LIN {X 0,Y 317.78,Z 749.574,A -85,B 0,C 180,E1 -15963.012,E2 -15963.012} C_VEL
LIN {X 0,Y 315.346,Z 742.44,A -85,B 0,C 180,E1 -15964.324,E2 -15964.324} C_VEL
LIN {X 0,Y 313.028,Z 732.738,A -85,B 0,C 180,E1 -15966.631,E2 -15966.631} C_VEL
LIN {X 0,Y 311.777,Z 725.359,A -85,B 0,C 180,E1 -15968.715,E2 -15968.715} C_VEL
LIN {X 0,Y 311.359,Z 724.12,A -85,B 0,C 180,E1 -15969.207,E2 -15969.207} C_VEL
LIN {X 0,Y 309.328,Z 721.332,A -85,B 0,C 180,E1 -15971.223,E2 -15971.223} C_VEL
LIN {X 0,Y 308.008,Z 719.093,A -85,B 0,C 180,E1 -15973.207,E2 -15973.207} C_VEL
LIN {X 0,Y 306.578,Z 717.561,A -85,B 0,C 180,E1 -15976.55,E2 -15976.55} C_VEL
LIN {X 0,Y 306.472,Z 717.374,A -85,B 0,C 180,E1 -15979.188,E2 -15979.188} C_VEL
LIN {X 0,Y 307.274,Z 718.36,A -85,B 0,C 180,E1 -15982.108,E2 -15982.108} C_VEL
LIN {X 0,Y 310.182,Z 720.574,A -85,B 0,C 180,E1 -15984.209,E2 -15984.209} C_VEL
LIN {X 0,Y 311.655,Z 723.597,A -85,B 0,C 180,E1 -15985.294,E2 -15985.294} C_VEL
LIN {X 0,Y 314.049,Z 725.859,A -85,B 0,C 180,E1 -15986.519,E2 -15986.519} C_VEL
LIN {X 0,Y 315.86,Z 729.038,A -85,B 0,C 180,E1 -15987.472,E2 -15987.472} C_VEL
LIN {X 0,Y 317.513,Z 730.978,A -85,B 0,C 180,E1 -15988.203,E2 -15988.203} C_VEL
LIN {X 0,Y 320.745,Z 736.046,A -85,B 0,C 180,E1 -15989.561,E2 -15989.561} C_VEL
LIN {X 0,Y 323.632,Z 740.623,A -85,B 0,C 180,E1 -15990.632,E2 -15990.632} C_VEL
LIN {X 0,Y 328.07,Z 748.441,A -85,B 0,C 180,E1 -15992.144,E2 -15992.144} C_VEL
LIN {X 0,Y 330.075,Z 752.544,A -85,B 0,C 180,E1 -15992.8,E2 -15992.8} C_VEL
LIN {X 0,Y 326.244,Z 796.508,A -85,B 0,C 180,E1 -15994.522,E2 -15994.522} C_VEL
LIN {X 0,Y 325.441,Z 812.458,A -85,B 0,C 180,E1 -15995.266,E2 -15995.266} C_VEL
LIN {X 0,Y 324.627,Z 823.18,A -85,B 0,C 180,E1 -15995.929,E2 -15995.929} C_VEL
LIN {X 0,Y 323.492,Z 834.349,A -85,B 0,C 180,E1 -15996.818,E2 -15996.818} C_VEL
LIN {X 0,Y 321.89,Z 846.494,A -85,B 0,C 180,E1 -15998.044,E2 -15998.044} C_VEL
LIN {X 0,Y 320.226,Z 856.26,A -85,B 0,C 180,E1 -15999.274,E2 -15999.274} C_VEL
LIN {X 0,Y 318.57,Z 865.22,A -85,B 0,C 180,E1 -16000.676,E2 -16000.676} C_VEL
LIN {X 0,Y 317.098,Z 871.96,A -85,B 0,C 180,E1 -16001.923,E2 -16001.923} C_VEL
LIN {X 0,Y 315.396,Z 879.003,A -85,B 0,C 180,E1 -16003.477,E2 -16003.477} C_VEL
LIN {X 0,Y 313.824,Z 884.946,A -85,B 0,C 180,E1 -16005.076,E2 -16005.076} C_VEL
LIN {X 0,Y 312.104,Z 890.624,A -85,B 0,C 180,E1 -16006.986,E2 -16006.986} C_VEL
LIN {X 0,Y 311.032,Z 893.718,A -85,B 0,C 180,E1 -16008.266,E2 -16008.266} C_VEL
LIN {X 0,Y 310.152,Z 896.329,A -85,B 0,C 180,E1 -16009.556,E2 -16009.556} C_VEL
LIN {X 0,Y 308.48,Z 899.873,A -85,B 0,C 180,E1 -16012.143,E2 -16012.143} C_VEL
LIN {X 0,Y 307.923,Z 901.043,A -85,B 0,C 180,E1 -16013.447,E2 -16013.447} C_VEL
LIN {X 0,Y 307.007,Z 901.892,A -85,B 0,C 180,E1 -16016.062,E2 -16016.062} C_VEL
LIN {X 0,Y 306.544,Z 901.716,A -85,B 0,C 180,E1 -16017.372,E2 -16017.372} C_VEL
LIN {X 0,Y 306.293,Z 901.04,A -85,B 0,C 180,E1 -16018.685,E2 -16018.685} C_VEL
LIN {X 0,Y 305.877,Z 899.917,A -85,B 0,C 180,E1 -16020,E2 -16020} C_VEL
LIN {X 0,Y 305.848,Z 898.443,A -85,B 0,C 180,E1 -16021.317,E2 -16021.317} C_VEL
LIN {X 0,Y 305.552,Z 895.298,A -85,B 0,C 180,E1 -16023.297,E2 -16023.297} C_VEL
LIN {X 0,Y 305.718,Z 891.017,A -85,B 0,C 180,E1 -16025.276,E2 -16025.276} C_VEL
LIN {X 0,Y 306.118,Z 885.522,A -85,B 0,C 180,E1 -16027.254,E2 -16027.254} C_VEL
LIN {X 0,Y 306.415,Z 879.941,A -85,B 0,C 180,E1 -16028.906,E2 -16028.906} C_VEL
LIN {X 0,Y 306.759,Z 873.225,A -85,B 0,C 180,E1 -16030.561,E2 -16030.561} C_VEL
LIN {X 0,Y 307.31,Z 865.158,A -85,B 0,C 180,E1 -16032.213,E2 -16032.213} C_VEL
LIN {X 0,Y 307.837,Z 856.481,A -85,B 0,C 180,E1 -16033.702,E2 -16033.702} C_VEL
LIN {X 0,Y 308.322,Z 848.553,A -85,B 0,C 180,E1 -16034.859,E2 -16034.859} C_VEL
LIN {X 0,Y 308.959,Z 839.214,A -85,B 0,C 180,E1 -16036.011,E2 -16036.011} C_VEL
LIN {X 0,Y 309.468,Z 829.618,A -85,B 0,C 180,E1 -16037.001,E2 -16037.001} C_VEL
LIN {X 0,Y 309.947,Z 818.852,A -85,B 0,C 180,E1 -16037.909,E2 -16037.909} C_VEL
LIN {X 0,Y 310.257,Z 809.036,A -85,B 0,C 180,E1 -16038.575,E2 -16038.575} C_VEL
LIN {X 0,Y 310.505,Z 798.799,A -85,B 0,C 180,E1 -16039.117,E2 -16039.117} C_VEL
LIN {X 0,Y 310.764,Z 784.432,A -85,B 0,C 180,E1 -16039.658,E2 -16039.658} C_VEL
LIN {X 0,Y 311.932,Z 734.903,A -85,B 0,C 180,E1 -16041.245,E2 -16041.245} C_VEL
LIN {X 0,Y 305.553,Z 714.421,A -85,B 0,C 180,E1 -16042.227,E2 -16042.227} C_VEL
LIN {X 0,Y 305.492,Z 714.43,A -85,B 0,C 180,E1 -16046.194,E2 -16046.194} C_VEL
LIN {X 0,Y 305.459,Z 714.438,A -85,B 0,C 180,E1 -16049.026,E2 -16049.026} C_VEL
LIN {X 0,Y 305.459,Z 714.434,A -85,B 0,C 180,E1 -16051.951,E2 -16051.951} C_VEL
LIN {X 0,Y 305.483,Z 714.432,A -85,B 0,C 180,E1 -16055.111,E2 -16055.111} C_VEL
LIN {X 0,Y 305.457,Z 714.434,A -85,B 0,C 180,E1 -16058.521,E2 -16058.521} C_VEL
LIN {X 0,Y 305.455,Z 714.432,A -85,B 0,C 180,E1 -16062.577,E2 -16062.577} C_VEL
LIN {X 0,Y 305.441,Z 714.431,A -85,B 0,C 180,E1 -16066.339,E2 -16066.339} C_VEL
LIN {X 0,Y 305.431,Z 714.433,A -85,B 0,C 180,E1 -16069.88,E2 -16069.88} C_VEL
LIN {X 0,Y 305.481,Z 714.427,A -85,B 0,C 180,E1 -16073.632,E2 -16073.632} C_VEL
LIN {X 0,Y 305.483,Z 714.427,A -85,B 0,C 180,E1 -16076.478,E2 -16076.478} C_VEL
LIN {X 0,Y 305.431,Z 714.436,A -85,B 0,C 180,E1 -16079.58,E2 -16079.58} C_VEL
LIN {X 0,Y 305.457,Z 714.431,A -85,B 0,C 180,E1 -16082.595,E2 -16082.595} C_VEL
LIN {X 0,Y 305.493,Z 714.428,A -85,B 0,C 180,E1 -16083.931,E2 -16083.931} C_VEL
LIN {X 0,Y 306.567,Z 717.417,A -85,B 0,C 180,E1 -16084.128,E2 -16084.128} C_VEL
LIN {X 0,Y 314.491,Z 733.858,A -85,B 0,C 180,E1 -16085.267,E2 -16085.267} C_VEL
LIN {X 0,Y 318.357,Z 742.756,A -85,B 0,C 180,E1 -16085.82,E2 -16085.82} C_VEL
LIN {X 0,Y 317.568,Z 789.63,A -85,B 0,C 180,E1 -16086.896,E2 -16086.896} C_VEL
LIN {X 0,Y 317.483,Z 803.278,A -85,B 0,C 180,E1 -16087.318,E2 -16087.318} C_VEL
LIN {X 0,Y 317.084,Z 815.616,A -85,B 0,C 180,E1 -16087.943,E2 -16087.943} C_VEL
LIN {X 0,Y 316.257,Z 828.425,A -85,B 0,C 180,E1 -16088.858,E2 -16088.858} C_VEL
LIN {X 0,Y 315.223,Z 840.006,A -85,B 0,C 180,E1 -16089.957,E2 -16089.957} C_VEL
LIN {X 0,Y 313.996,Z 850.475,A -85,B 0,C 180,E1 -16091.224,E2 -16091.224} C_VEL
LIN {X 0,Y 312.703,Z 860.073,A -85,B 0,C 180,E1 -16092.667,E2 -16092.667} C_VEL
LIN {X 0,Y 311.526,Z 868.767,A -85,B 0,C 180,E1 -16094.285,E2 -16094.285} C_VEL
LIN {X 0,Y 310.053,Z 877.271,A -85,B 0,C 180,E1 -16096.223,E2 -16096.223} C_VEL
LIN {X 0,Y 308.81,Z 884.034,A -85,B 0,C 180,E1 -16098.173,E2 -16098.173} C_VEL
LIN {X 0,Y 308.073,Z 889.399,A -85,B 0,C 180,E1 -16100.14,E2 -16100.14} C_VEL
LIN {X 0,Y 307.587,Z 892.335,A -85,B 0,C 180,E1 -16101.451,E2 -16101.451} C_VEL
LIN {X 0,Y 306.655,Z 895.896,A -85,B 0,C 180,E1 -16103.412,E2 -16103.412} C_VEL
LIN {X 0,Y 306.29,Z 897.719,A -85,B 0,C 180,E1 -16104.725,E2 -16104.725} C_VEL
LIN {X 0,Y 306.079,Z 900.031,A -85,B 0,C 180,E1 -16107.359,E2 -16107.359} C_VEL
LIN {X 0,Y 305.857,Z 900.872,A -85,B 0,C 180,E1 -16109.991,E2 -16109.991} C_VEL
LIN {X 0,Y 306.079,Z 900.108,A -85,B 0,C 180,E1 -16112.623,E2 -16112.623} C_VEL
LIN {X 0,Y 306.272,Z 897.878,A -85,B 0,C 180,E1 -16115.257,E2 -16115.257} C_VEL
LIN {X 0,Y 306.892,Z 895.061,A -85,B 0,C 180,E1 -16117.227,E2 -16117.227} C_VEL
LIN {X 0,Y 307.753,Z 891.234,A -85,B 0,C 180,E1 -16119.189,E2 -16119.189} C_VEL
LIN {X 0,Y 308.611,Z 885.762,A -85,B 0,C 180,E1 -16121.358,E2 -16121.358} C_VEL
LIN {X 0,Y 309.801,Z 878.949,A -85,B 0,C 180,E1 -16123.436,E2 -16123.436} C_VEL
LIN {X 0,Y 311.214,Z 870.92,A -85,B 0,C 180,E1 -16125.377,E2 -16125.377} C_VEL
LIN {X 0,Y 312.441,Z 862.701,A -85,B 0,C 180,E1 -16126.993,E2 -16126.993} C_VEL
LIN {X 0,Y 313.765,Z 852.531,A -85,B 0,C 180,E1 -16128.603,E2 -16128.603} C_VEL
LIN {X 0,Y 315.084,Z 842.061,A -85,B 0,C 180,E1 -16129.92,E2 -16129.92} C_VEL
LIN {X 0,Y 316.183,Z 830.793,A -85,B 0,C 180,E1 -16131.048,E2 -16131.048} C_VEL
LIN {X 0,Y 317.074,Z 818.868,A -85,B 0,C 180,E1 -16131.954,E2 -16131.954} C_VEL
LIN {X 0,Y 317.491,Z 806.497,A -85,B 0,C 180,E1 -16132.646,E2 -16132.646} C_VEL
LIN {X 0,Y 317.657,Z 795.086,A -85,B 0,C 180,E1 -16133.069,E2 -16133.069} C_VEL
LIN {X 0,Y 318.132,Z 758.842,A -85,B 0,C 180,E1 -16133.922,E2 -16133.922} C_VEL
LIN {X 0,Y 318.417,Z 742.883,A -85,B 0,C 180,E1 -16134.287,E2 -16134.287} C_VEL
LIN {X 0,Y 310.461,Z 725.118,A -85,B 0,C 180,E1 -16135.431,E2 -16135.431} C_VEL
LIN {X 0,Y 305.739,Z 715.497,A -85,B 0,C 180,E1 -16136.119,E2 -16136.119} C_VEL
LIN {X 0,Y 305.504,Z 714.422,A -85,B 0,C 180,E1 -16136.21,E2 -16136.21} C_VEL
LIN {X 0,Y 305.424,Z 714.435,A -85,B 0,C 180,E1 -16140.188,E2 -16140.188} C_VEL
LIN {X 0,Y 305.433,Z 714.435,A -85,B 0,C 180,E1 -16144.069,E2 -16144.069} C_VEL
LIN {X 0,Y 305.435,Z 714.436,A -85,B 0,C 180,E1 -16145.905,E2 -16145.905} C_VEL
LIN {X 0,Y 304.811,Z 714.517,A -85,B 0,C 180,E1 -16147.006,E2 -16147.006} C_VEL
LIN {X 0,Y 301.976,Z 714.877,A -85,B 0,C 180,E1 -16148.797,E2 -16148.797} C_VEL
LIN {X 0,Y 299.539,Z 715.18,A -85,B 0,C 180,E1 -16150.251,E2 -16150.251} C_VEL
LIN {X 0,Y 298.48,Z 715.31,A -85,B 0,C 180,E1 -16151.377,E2 -16151.377} C_VEL
LIN {X 0,Y 298.389,Z 715.314,A -85,B 0,C 180,E1 -16151.758,E2 -16151.758} C_VEL
LIN {X 0,Y 298.446,Z 715.285,A -85,B 0,C 180,E1 -16155.052,E2 -16155.052} C_VEL
LIN {X 0,Y 298.407,Z 715.316,A -85,B 0,C 180,E1 -16158.89,E2 -16158.89} C_VEL
LIN {X 0,Y 298.415,Z 715.312,A -85,B 0,C 180,E1 -16163.18,E2 -16163.18} C_VEL
LIN {X 0,Y 298.343,Z 715.317,A -85,B 0,C 180,E1 -16167.193,E2 -16167.193} C_VEL
LIN {X 0,Y 298.376,Z 715.306,A -85,B 0,C 180,E1 -16170.609,E2 -16170.609} C_VEL
LIN {X 0,Y 298.421,Z 715.31,A -85,B 0,C 180,E1 -16173.471,E2 -16173.471} C_VEL
LIN {X 0,Y 298.373,Z 715.308,A -85,B 0,C 180,E1 -16176.694,E2 -16176.694} C_VEL
LIN {X 0,Y 298.476,Z 715.3,A -85,B 0,C 180,E1 -16180.752,E2 -16180.752} C_VEL
LIN {X 0,Y 298.528,Z 715.3,A -85,B 0,C 180,E1 -16184.991,E2 -16184.991} C_VEL
LIN {X 0,Y 298.527,Z 715.286,A -85,B 0,C 180,E1 -16189.144,E2 -16189.144} C_VEL
LIN {X 0,Y 298.683,Z 715.28,A -85,B 0,C 180,E1 -16191.884,E2 -16191.884} C_VEL
LIN {X 0,Y 298.595,Z 715.288,A -85,B 0,C 180,E1 -16194.598,E2 -16194.598} C_VEL
LIN {X 0,Y 298.861,Z 715.26,A -85,B 0,C 180,E1 -16198.652,E2 -16198.652} C_VEL
LIN {X 0,Y 298.861,Z 715.253,A -85,B 0,C 180,E1 -16201.347,E2 -16201.347} C_VEL
LIN {X 0,Y 298.596,Z 715.296,A -85,B 0,C 180,E1 -16205.402,E2 -16205.402} C_VEL
LIN {X 0,Y 298.683,Z 715.274,A -85,B 0,C 180,E1 -16208.116,E2 -16208.116} C_VEL
LIN {X 0,Y 298.488,Z 715.304,A -85,B 0,C 180,E1 -16212.234,E2 -16212.234} C_VEL
LIN {X 0,Y 298.521,Z 715.301,A -85,B 0,C 180,E1 -16215.198,E2 -16215.198} C_VEL
LIN {X 0,Y 298.462,Z 715.305,A -85,B 0,C 180,E1 -16219.248,E2 -16219.248} C_VEL
LIN {X 0,Y 298.395,Z 715.317,A -85,B 0,C 180,E1 -16223.603,E2 -16223.603} C_VEL
LIN {X 0,Y 298.427,Z 715.303,A -85,B 0,C 180,E1 -16226.58,E2 -16226.58} C_VEL
LIN {X 0,Y 298.365,Z 715.313,A -85,B 0,C 180,E1 -16229.647,E2 -16229.647} C_VEL
LIN {X 0,Y 298.343,Z 715.32,A -85,B 0,C 180,E1 -16232.807,E2 -16232.807} C_VEL
LIN {X 0,Y 298.415,Z 715.309,A -85,B 0,C 180,E1 -16236.82,E2 -16236.82} C_VEL
LIN {X 0,Y 298.407,Z 715.314,A -85,B 0,C 180,E1 -16241.258,E2 -16241.258} C_VEL
LIN {X 0,Y 298.446,Z 715.308,A -85,B 0,C 180,E1 -16245.069,E2 -16245.069} C_VEL
LIN {X 0,Y 298.414,Z 715.312,A -85,B 0,C 180,E1 -16248.907,E2 -16248.907} C_VEL
LIN {X 0,Y 298.416,Z 715.345,A -85,B 0,C 180,E1 -16249.765,E2 -16249.765} C_VEL
LIN {X 0,Y 301.883,Z 728.539,A -85,B 0,C 180,E1 -16253.434,E2 -16253.434} C_VEL
LIN {X 0,Y 304.482,Z 739.897,A -85,B 0,C 180,E1 -16256.374,E2 -16256.374} C_VEL
LIN {X 0,Y 306.355,Z 749.348,A -85,B 0,C 180,E1 -16258.703,E2 -16258.703} C_VEL
LIN {X 0,Y 303.364,Z 769.628,A -85,B 0,C 180,E1 -16263.081,E2 -16263.081} C_VEL
LIN {X 0,Y 307.305,Z 801.463,A -85,B 0,C 180,E1 -16264.256,E2 -16264.256} C_VEL
LIN {X 0,Y 310.222,Z 833.466,A -85,B 0,C 180,E1 -16265.3,E2 -16265.3} C_VEL
LIN {X 0,Y 308.939,Z 881.214,A -85,B 0,C 180,E1 -16266.418,E2 -16266.418} C_VEL
LIN {X 0,Y 308.109,Z 894.367,A -85,B 0,C 180,E1 -16266.973,E2 -16266.973} C_VEL
LIN {X 0,Y 306.749,Z 907.617,A -85,B 0,C 180,E1 -16267.799,E2 -16267.799} C_VEL
LIN {X 0,Y 305.001,Z 920.376,A -85,B 0,C 180,E1 -16268.908,E2 -16268.908} C_VEL
LIN {X 0,Y 303.313,Z 931.755,A -85,B 0,C 180,E1 -16270.203,E2 -16270.203} C_VEL
LIN {X 0,Y 301.654,Z 942.042,A -85,B 0,C 180,E1 -16271.678,E2 -16271.678} C_VEL
LIN {X 0,Y 300.261,Z 951.365,A -85,B 0,C 180,E1 -16273.348,E2 -16273.348} C_VEL
LIN {X 0,Y 299.218,Z 957.951,A -85,B 0,C 180,E1 -16274.754,E2 -16274.754} C_VEL
LIN {X 0,Y 298.26,Z 965.572,A -85,B 0,C 180,E1 -16276.728,E2 -16276.728} C_VEL
LIN {X 0,Y 297.557,Z 972.9,A -85,B 0,C 180,E1 -16279.118,E2 -16279.118} C_VEL
LIN {X 0,Y 297.357,Z 977.823,A -85,B 0,C 180,E1 -16281.173,E2 -16281.173} C_VEL
LIN {X 0,Y 297.456,Z 981.629,A -85,B 0,C 180,E1 -16283.225,E2 -16283.225} C_VEL
LIN {X 0,Y 297.577,Z 983.601,A -85,B 0,C 180,E1 -16284.589,E2 -16284.589} C_VEL
LIN {X 0,Y 297.805,Z 985.098,A -85,B 0,C 180,E1 -16285.949,E2 -16285.949} C_VEL
LIN {X 0,Y 297.879,Z 986.153,A -85,B 0,C 180,E1 -16287.305,E2 -16287.305} C_VEL
LIN {X 0,Y 297.996,Z 986.804,A -85,B 0,C 180,E1 -16288.658,E2 -16288.658} C_VEL
LIN {X 0,Y 298.112,Z 987.041,A -85,B 0,C 180,E1 -16290.009,E2 -16290.009} C_VEL
LIN {X 0,Y 297.996,Z 986.79,A -85,B 0,C 180,E1 -16291.36,E2 -16291.36} C_VEL
LIN {X 0,Y 297.88,Z 986.129,A -85,B 0,C 180,E1 -16292.713,E2 -16292.713} C_VEL
LIN {X 0,Y 297.8,Z 985.064,A -85,B 0,C 180,E1 -16294.069,E2 -16294.069} C_VEL
LIN {X 0,Y 297.555,Z 983.55,A -85,B 0,C 180,E1 -16295.43,E2 -16295.43} C_VEL
LIN {X 0,Y 297.375,Z 980.431,A -85,B 0,C 180,E1 -16297.477,E2 -16297.477} C_VEL
LIN {X 0,Y 297.411,Z 976.25,A -85,B 0,C 180,E1 -16299.53,E2 -16299.53} C_VEL
LIN {X 0,Y 297.908,Z 969.561,A -85,B 0,C 180,E1 -16302.267,E2 -16302.267} C_VEL
LIN {X 0,Y 298.553,Z 964.531,A -85,B 0,C 180,E1 -16303.971,E2 -16303.971} C_VEL
LIN {X 0,Y 299.246,Z 959.384,A -85,B 0,C 180,E1 -16305.465,E2 -16305.465} C_VEL
LIN {X 0,Y 300.95,Z 951.553,A -85,B 0,C 180,E1 -16307.33,E2 -16307.33} C_VEL
LIN {X 0,Y 302.197,Z 945.189,A -85,B 0,C 180,E1 -16308.657,E2 -16308.657} C_VEL
LIN {X 0,Y 304.243,Z 935.751,A -85,B 0,C 180,E1 -16310.281,E2 -16310.281} C_VEL
LIN {X 0,Y 306.431,Z 925.609,A -85,B 0,C 180,E1 -16311.713,E2 -16311.713} C_VEL
LIN {X 0,Y 308.42,Z 916.446,A -85,B 0,C 180,E1 -16312.799,E2 -16312.799} C_VEL
LIN {X 0,Y 310.592,Z 905.498,A -85,B 0,C 180,E1 -16313.866,E2 -16313.866} C_VEL
LIN {X 0,Y 312.674,Z 893.979,A -85,B 0,C 180,E1 -16314.756,E2 -16314.756} C_VEL
LIN {X 0,Y 314.473,Z 882.009,A -85,B 0,C 180,E1 -16315.488,E2 -16315.488} C_VEL
LIN {X 0,Y 315.97,Z 869.576,A -85,B 0,C 180,E1 -16316.066,E2 -16316.066} C_VEL
LIN {X 0,Y 318.92,Z 833.781,A -85,B 0,C 180,E1 -16317.446,E2 -16317.446} C_VEL
LIN {X 0,Y 318.912,Z 810.916,A -85,B 0,C 180,E1 -16318.73,E2 -16318.73} C_VEL
LIN {X 0,Y 318.007,Z 792.559,A -85,B 0,C 180,E1 -16320.021,E2 -16320.021} C_VEL
LIN {X 0,Y 316.783,Z 775.824,A -85,B 0,C 180,E1 -16321.396,E2 -16321.396} C_VEL
LIN {X 0,Y 315.684,Z 763.889,A -85,B 0,C 180,E1 -16322.517,E2 -16322.517} C_VEL
LIN {X 0,Y 315.141,Z 758.222,A -85,B 0,C 180,E1 -16323.103,E2 -16323.103} C_VEL
LIN {X 0,Y 313.114,Z 751.058,A -85,B 0,C 180,E1 -16324.284,E2 -16324.284} C_VEL
LIN {X 0,Y 309.302,Z 739.293,A -85,B 0,C 180,E1 -16326.775,E2 -16326.775} C_VEL
LIN {X 0,Y 307.953,Z 731.002,A -85,B 0,C 180,E1 -16329.11,E2 -16329.11} C_VEL
LIN {X 0,Y 306.237,Z 728.311,A -85,B 0,C 180,E1 -16330.77,E2 -16330.77} C_VEL
LIN {X 0,Y 304.964,Z 726.058,A -85,B 0,C 180,E1 -16332.485,E2 -16332.485} C_VEL
LIN {X 0,Y 303.86,Z 724.705,A -85,B 0,C 180,E1 -16334.192,E2 -16334.192} C_VEL
LIN {X 0,Y 302.724,Z 723.437,A -85,B 0,C 180,E1 -16337.681,E2 -16337.681} C_VEL
LIN {X 0,Y 302.862,Z 723.49,A -85,B 0,C 180,E1 -16338.774,E2 -16338.774} C_VEL
LIN {X 0,Y 305.23,Z 725.008,A -85,B 0,C 180,E1 -16341.798,E2 -16341.798} C_VEL
LIN {X 0,Y 307.862,Z 727.156,A -85,B 0,C 180,E1 -16343.868,E2 -16343.868} C_VEL
LIN {X 0,Y 309.371,Z 730.118,A -85,B 0,C 180,E1 -16345.004,E2 -16345.004} C_VEL
LIN {X 0,Y 311.415,Z 732.252,A -85,B 0,C 180,E1 -16346.13,E2 -16346.13} C_VEL
LIN {X 0,Y 313.525,Z 735.695,A -85,B 0,C 180,E1 -16347.276,E2 -16347.276} C_VEL
LIN {X 0,Y 314.806,Z 737.475,A -85,B 0,C 180,E1 -16347.88,E2 -16347.88} C_VEL
LIN {X 0,Y 317.575,Z 741.889,A -85,B 0,C 180,E1 -16349.106,E2 -16349.106} C_VEL
LIN {X 0,Y 321.106,Z 747.72,A -85,B 0,C 180,E1 -16350.494,E2 -16350.494} C_VEL
LIN {X 0,Y 325.184,Z 755.627,A -85,B 0,C 180,E1 -16351.967,E2 -16351.967} C_VEL
LIN {X 0,Y 321.393,Z 795.17,A -85,B 0,C 180,E1 -16353.555,E2 -16353.555} C_VEL
LIN {X 0,Y 320.302,Z 812.935,A -85,B 0,C 180,E1 -16354.399,E2 -16354.399} C_VEL
LIN {X 0,Y 319.306,Z 824.586,A -85,B 0,C 180,E1 -16355.136,E2 -16355.136} C_VEL
LIN {X 0,Y 317.983,Z 836.68,A -85,B 0,C 180,E1 -16356.122,E2 -16356.122} C_VEL
LIN {X 0,Y 316.114,Z 849.232,A -85,B 0,C 180,E1 -16357.449,E2 -16357.449} C_VEL
LIN {X 0,Y 314.33,Z 858.649,A -85,B 0,C 180,E1 -16358.695,E2 -16358.695} C_VEL
LIN {X 0,Y 312.357,Z 868.303,A -85,B 0,C 180,E1 -16360.275,E2 -16360.275} C_VEL
LIN {X 0,Y 310.799,Z 874.787,A -85,B 0,C 180,E1 -16361.544,E2 -16361.544} C_VEL
LIN {X 0,Y 309.351,Z 880.337,A -85,B 0,C 180,E1 -16362.822,E2 -16362.822} C_VEL
LIN {X 0,Y 307.636,Z 886.169,A -85,B 0,C 180,E1 -16364.429,E2 -16364.429} C_VEL
LIN {X 0,Y 306.085,Z 891.029,A -85,B 0,C 180,E1 -16366.049,E2 -16366.049} C_VEL
LIN {X 0,Y 304.914,Z 894.333,A -85,B 0,C 180,E1 -16367.352,E2 -16367.352} C_VEL
LIN {X 0,Y 303.401,Z 898.107,A -85,B 0,C 180,E1 -16369.321,E2 -16369.321} C_VEL
LIN {X 0,Y 302.482,Z 899.997,A -85,B 0,C 180,E1 -16370.64,E2 -16370.64} C_VEL
LIN {X 0,Y 301.035,Z 902.452,A -85,B 0,C 180,E1 -16373.297,E2 -16373.297} C_VEL
LIN {X 0,Y 300.489,Z 903.002,A -85,B 0,C 180,E1 -16374.632,E2 -16374.632} C_VEL
LIN {X 0,Y 300.054,Z 903.151,A -85,B 0,C 180,E1 -16375.971,E2 -16375.971} C_VEL
LIN {X 0,Y 299.548,Z 902.829,A -85,B 0,C 180,E1 -16377.311,E2 -16377.311} C_VEL
LIN {X 0,Y 299.285,Z 902.06,A -85,B 0,C 180,E1 -16378.654,E2 -16378.654} C_VEL
LIN {X 0,Y 298.85,Z 900.815,A -85,B 0,C 180,E1 -16380,E2 -16380} C_VEL
LIN {X 0,Y 298.67,Z 898.18,A -85,B 0,C 180,E1 -16382.023,E2 -16382.023} C_VEL
LIN {X 0,Y 298.424,Z 894.513,A -85,B 0,C 180,E1 -16384.051,E2 -16384.051} C_VEL
LIN {X 0,Y 298.84,Z 889.667,A -85,B 0,C 180,E1 -16386.075,E2 -16386.075} C_VEL
LIN {X 0,Y 299.133,Z 883.582,A -85,B 0,C 180,E1 -16388.104,E2 -16388.104} C_VEL
LIN {X 0,Y 299.653,Z 874.693,A -85,B 0,C 180,E1 -16390.439,E2 -16390.439} C_VEL
LIN {X 0,Y 300.197,Z 866.519,A -85,B 0,C 180,E1 -16392.164,E2 -16392.164} C_VEL
LIN {X 0,Y 300.738,Z 857.905,A -85,B 0,C 180,E1 -16393.687,E2 -16393.687} C_VEL
LIN {X 0,Y 301.201,Z 850.055,A -85,B 0,C 180,E1 -16394.872,E2 -16394.872} C_VEL
LIN {X 0,Y 301.876,Z 840.796,A -85,B 0,C 180,E1 -16396.049,E2 -16396.049} C_VEL
LIN {X 0,Y 302.383,Z 831.301,A -85,B 0,C 180,E1 -16397.064,E2 -16397.064} C_VEL
LIN {X 0,Y 302.874,Z 820.89,A -85,B 0,C 180,E1 -16397.976,E2 -16397.976} C_VEL
LIN {X 0,Y 303.218,Z 810.82,A -85,B 0,C 180,E1 -16398.689,E2 -16398.689} C_VEL
LIN {X 0,Y 303.49,Z 800.303,A -85,B 0,C 180,E1 -16399.268,E2 -16399.268} C_VEL
LIN {X 0,Y 303.747,Z 786.177,A -85,B 0,C 180,E1 -16399.823,E2 -16399.823} C_VEL
LIN {X 0,Y 304.999,Z 736.395,A -85,B 0,C 180,E1 -16401.463,E2 -16401.463} C_VEL
LIN {X 0,Y 298.494,Z 715.302,A -85,B 0,C 180,E1 -16402.511,E2 -16402.511} C_VEL
LIN {X 0,Y 298.432,Z 715.312,A -85,B 0,C 180,E1 -16406.58,E2 -16406.58} C_VEL
LIN {X 0,Y 298.385,Z 715.315,A -85,B 0,C 180,E1 -16409.645,E2 -16409.645} C_VEL
LIN {X 0,Y 298.416,Z 715.313,A -85,B 0,C 180,E1 -16412.798,E2 -16412.798} C_VEL
LIN {X 0,Y 298.426,Z 715.307,A -85,B 0,C 180,E1 -16416.069,E2 -16416.069} C_VEL
LIN {X 0,Y 298.397,Z 715.312,A -85,B 0,C 180,E1 -16419.488,E2 -16419.488} C_VEL
LIN {X 0,Y 298.391,Z 715.313,A -85,B 0,C 180,E1 -16423.093,E2 -16423.093} C_VEL
LIN {X 0,Y 298.391,Z 715.31,A -85,B 0,C 180,E1 -16426.91,E2 -16426.91} C_VEL
LIN {X 0,Y 298.406,Z 715.308,A -85,B 0,C 180,E1 -16431.006,E2 -16431.006} C_VEL
LIN {X 0,Y 298.423,Z 715.306,A -85,B 0,C 180,E1 -16433.923,E2 -16433.923} C_VEL
LIN {X 0,Y 298.411,Z 715.308,A -85,B 0,C 180,E1 -16437.194,E2 -16437.194} C_VEL
LIN {X 0,Y 298.38,Z 715.312,A -85,B 0,C 180,E1 -16440.633,E2 -16440.633} C_VEL
LIN {X 0,Y 298.425,Z 715.311,A -85,B 0,C 180,E1 -16443.271,E2 -16443.271} C_VEL
LIN {X 0,Y 299.407,Z 718.12,A -85,B 0,C 180,E1 -16443.449,E2 -16443.449} C_VEL
LIN {X 0,Y 306.959,Z 733.357,A -85,B 0,C 180,E1 -16444.574,E2 -16444.574} C_VEL
LIN {X 0,Y 311.92,Z 744.69,A -85,B 0,C 180,E1 -16445.31,E2 -16445.31} C_VEL
LIN {X 0,Y 311.096,Z 789.997,A -85,B 0,C 180,E1 -16446.37,E2 -16446.37} C_VEL
LIN {X 0,Y 310.99,Z 804.558,A -85,B 0,C 180,E1 -16446.828,E2 -16446.828} C_VEL
LIN {X 0,Y 310.578,Z 816.628,A -85,B 0,C 180,E1 -16447.456,E2 -16447.456} C_VEL
LIN {X 0,Y 309.712,Z 829.435,A -85,B 0,C 180,E1 -16448.389,E2 -16448.389} C_VEL
LIN {X 0,Y 308.63,Z 841.014,A -85,B 0,C 180,E1 -16449.51,E2 -16449.51} C_VEL
LIN {X 0,Y 307.351,Z 851.482,A -85,B 0,C 180,E1 -16450.802,E2 -16450.802} C_VEL
LIN {X 0,Y 306.001,Z 861.079,A -85,B 0,C 180,E1 -16452.275,E2 -16452.275} C_VEL
LIN {X 0,Y 304.767,Z 869.773,A -85,B 0,C 180,E1 -16453.927,E2 -16453.927} C_VEL
LIN {X 0,Y 303.232,Z 878.276,A -85,B 0,C 180,E1 -16455.907,E2 -16455.907} C_VEL
LIN {X 0,Y 301.935,Z 885.038,A -85,B 0,C 180,E1 -16457.899,E2 -16457.899} C_VEL
LIN {X 0,Y 301.151,Z 890.403,A -85,B 0,C 180,E1 -16459.911,E2 -16459.911} C_VEL
LIN {X 0,Y 300.64,Z 893.339,A -85,B 0,C 180,E1 -16461.252,E2 -16461.252} C_VEL
LIN {X 0,Y 299.675,Z 896.899,A -85,B 0,C 180,E1 -16463.257,E2 -16463.257} C_VEL
LIN {X 0,Y 299.292,Z 898.722,A -85,B 0,C 180,E1 -16464.602,E2 -16464.602} C_VEL
LIN {X 0,Y 299.06,Z 901.033,A -85,B 0,C 180,E1 -16467.297,E2 -16467.297} C_VEL
LIN {X 0,Y 298.83,Z 901.875,A -85,B 0,C 180,E1 -16469.991,E2 -16469.991} C_VEL
LIN {X 0,Y 299.059,Z 901.11,A -85,B 0,C 180,E1 -16472.685,E2 -16472.685} C_VEL
LIN {X 0,Y 299.273,Z 898.88,A -85,B 0,C 180,E1 -16475.381,E2 -16475.381} C_VEL
LIN {X 0,Y 299.922,Z 896.063,A -85,B 0,C 180,E1 -16477.395,E2 -16477.395} C_VEL
LIN {X 0,Y 300.818,Z 892.235,A -85,B 0,C 180,E1 -16479.403,E2 -16479.403} C_VEL
LIN {X 0,Y 301.724,Z 886.763,A -85,B 0,C 180,E1 -16481.621,E2 -16481.621} C_VEL
LIN {X 0,Y 302.97,Z 879.95,A -85,B 0,C 180,E1 -16483.745,E2 -16483.745} C_VEL
LIN {X 0,Y 304.444,Z 871.92,A -85,B 0,C 180,E1 -16485.728,E2 -16485.728} C_VEL
LIN {X 0,Y 305.727,Z 863.701,A -85,B 0,C 180,E1 -16487.378,E2 -16487.378} C_VEL
LIN {X 0,Y 307.112,Z 853.53,A -85,B 0,C 180,E1 -16489.022,E2 -16489.022} C_VEL
LIN {X 0,Y 308.486,Z 843.059,A -85,B 0,C 180,E1 -16490.365,E2 -16490.365} C_VEL
LIN {X 0,Y 309.633,Z 831.789,A -85,B 0,C 180,E1 -16491.515,E2 -16491.515} C_VEL
LIN {X 0,Y 310.565,Z 819.862,A -85,B 0,C 180,E1 -16492.439,E2 -16492.439} C_VEL
LIN {X 0,Y 310.998,Z 807.714,A -85,B 0,C 180,E1 -16493.135,E2 -16493.135} C_VEL
LIN {X 0,Y 311.158,Z 796.736,A -85,B 0,C 180,E1 -16493.56,E2 -16493.56} C_VEL
LIN {X 0,Y 311.792,Z 754.155,A -85,B 0,C 180,E1 -16494.581,E2 -16494.581} C_VEL
LIN {X 0,Y 311.98,Z 744.708,A -85,B 0,C 180,E1 -16494.801,E2 -16494.801} C_VEL
LIN {X 0,Y 303.617,Z 726.251,A -85,B 0,C 180,E1 -16496.044,E2 -16496.044} C_VEL
LIN {X 0,Y 298.674,Z 716.431,A -85,B 0,C 180,E1 -16496.79,E2 -16496.79} C_VEL
LIN {X 0,Y 298.443,Z 715.305,A -85,B 0,C 180,E1 -16496.879,E2 -16496.879} C_VEL
LIN {X 0,Y 298.39,Z 715.312,A -85,B 0,C 180,E1 -16499.632,E2 -16499.632} C_VEL
LIN {X 0,Y 298.365,Z 715.32,A -85,B 0,C 180,E1 -16502.791,E2 -16502.791} C_VEL
LIN {X 0,Y 298.431,Z 715.306,A -85,B 0,C 180,E1 -16506.803,E2 -16506.803} C_VEL
LIN {X 0,Y 298.415,Z 715.317,A -85,B 0,C 180,E1 -16511.241,E2 -16511.241} C_VEL
LIN {X 0,Y 298.389,Z 715.314,A -85,B 0,C 180,E1 -16511.758,E2 -16511.758} C_VEL
LIN {X 0,Y 297.713,Z 715.4,A -85,B 0,C 180,E1 -16512.886,E2 -16512.886} C_VEL
LIN {X 0,Y 294.88,Z 715.74,A -85,B 0,C 180,E1 -16514.722,E2 -16514.722} C_VEL
LIN {X 0,Y 292.478,Z 716.041,A -85,B 0,C 180,E1 -16516.212,E2 -16516.212} C_VEL
LIN {X 0,Y 291.436,Z 716.176,A -85,B 0,C 180,E1 -16517.366,E2 -16517.366} C_VEL
LIN {X 0,Y 291.345,Z 716.19,A -85,B 0,C 180,E1 -16517.757,E2 -16517.757} C_VEL
LIN {X 0,Y 291.329,Z 716.19,A -85,B 0,C 180,E1 -16521.154,E2 -16521.154} C_VEL
LIN {X 0,Y 291.334,Z 716.191,A -85,B 0,C 180,E1 -16524.622,E2 -16524.622} C_VEL
LIN {X 0,Y 291.321,Z 716.196,A -85,B 0,C 180,E1 -16527.944,E2 -16527.944} C_VEL
LIN {X 0,Y 291.325,Z 716.184,A -85,B 0,C 180,E1 -16531.152,E2 -16531.152} C_VEL
LIN {X 0,Y 291.356,Z 716.192,A -85,B 0,C 180,E1 -16534.266,E2 -16534.266} C_VEL
LIN {X 0,Y 291.32,Z 716.189,A -85,B 0,C 180,E1 -16537.294,E2 -16537.294} C_VEL
LIN {X 0,Y 291.397,Z 716.187,A -85,B 0,C 180,E1 -16540.266,E2 -16540.266} C_VEL
LIN {X 0,Y 291.477,Z 716.174,A -85,B 0,C 180,E1 -16544.631,E2 -16544.631} C_VEL
LIN {X 0,Y 291.471,Z 716.165,A -85,B 0,C 180,E1 -16548.878,E2 -16548.878} C_VEL
LIN {X 0,Y 291.636,Z 716.158,A -85,B 0,C 180,E1 -16551.686,E2 -16551.686} C_VEL
LIN {X 0,Y 291.565,Z 716.165,A -85,B 0,C 180,E1 -16554.467,E2 -16554.467} C_VEL
LIN {X 0,Y 291.828,Z 716.135,A -85,B 0,C 180,E1 -16558.62,E2 -16558.62} C_VEL
LIN {X 0,Y 291.828,Z 716.129,A -85,B 0,C 180,E1 -16561.38,E2 -16561.38} C_VEL
LIN {X 0,Y 291.565,Z 716.171,A -85,B 0,C 180,E1 -16565.533,E2 -16565.533} C_VEL
LIN {X 0,Y 291.636,Z 716.152,A -85,B 0,C 180,E1 -16568.314,E2 -16568.314} C_VEL
LIN {X 0,Y 291.455,Z 716.18,A -85,B 0,C 180,E1 -16572.534,E2 -16572.534} C_VEL
LIN {X 0,Y 291.475,Z 716.181,A -85,B 0,C 180,E1 -16575.381,E2 -16575.381} C_VEL
LIN {X 0,Y 291.39,Z 716.178,A -85,B 0,C 180,E1 -16579.879,E2 -16579.879} C_VEL
LIN {X 0,Y 291.337,Z 716.191,A -85,B 0,C 180,E1 -16584.211,E2 -16584.211} C_VEL
LIN {X 0,Y 291.363,Z 716.186,A -85,B 0,C 180,E1 -16587.278,E2 -16587.278} C_VEL
LIN {X 0,Y 291.283,Z 716.192,A -85,B 0,C 180,E1 -16590.443,E2 -16590.443} C_VEL
LIN {X 0,Y 291.292,Z 716.196,A -85,B 0,C 180,E1 -16593.705,E2 -16593.705} C_VEL
LIN {X 0,Y 291.348,Z 716.186,A -85,B 0,C 180,E1 -16597.267,E2 -16597.267} C_VEL
LIN {X 0,Y 291.354,Z 716.187,A -85,B 0,C 180,E1 -16600.639,E2 -16600.639} C_VEL
LIN {X 0,Y 291.363,Z 716.191,A -85,B 0,C 180,E1 -16604.388,E2 -16604.388} C_VEL
LIN {X 0,Y 291.349,Z 716.186,A -85,B 0,C 180,E1 -16608.4,E2 -16608.4} C_VEL
LIN {X 0,Y 291.399,Z 716.357,A -85,B 0,C 180,E1 -16609.151,E2 -16609.151} C_VEL
LIN {X 0,Y 294.076,Z 726.387,A -85,B 0,C 180,E1 -16612.06,E2 -16612.06} C_VEL
LIN {X 0,Y 297.078,Z 738.746,A -85,B 0,C 180,E1 -16615.419,E2 -16615.419} C_VEL
LIN {X 0,Y 299.369,Z 749.953,A -85,B 0,C 180,E1 -16618.283,E2 -16618.283} C_VEL
LIN {X 0,Y 298.875,Z 754.274,A -85,B 0,C 180,E1 -16619.252,E2 -16619.252} C_VEL
LIN {X 0,Y 296.704,Z 768.599,A -85,B 0,C 180,E1 -16622.431,E2 -16622.431} C_VEL
LIN {X 0,Y 300.55,Z 799.285,A -85,B 0,C 180,E1 -16623.605,E2 -16623.605} C_VEL
LIN {X 0,Y 303.709,Z 833.262,A -85,B 0,C 180,E1 -16624.754,E2 -16624.754} C_VEL
LIN {X 0,Y 302.456,Z 880.217,A -85,B 0,C 180,E1 -16625.881,E2 -16625.881} C_VEL
LIN {X 0,Y 301.528,Z 893.354,A -85,B 0,C 180,E1 -16626.441,E2 -16626.441} C_VEL
LIN {X 0,Y 300.164,Z 906.606,A -85,B 0,C 180,E1 -16627.285,E2 -16627.285} C_VEL
LIN {X 0,Y 298.381,Z 919.367,A -85,B 0,C 180,E1 -16628.417,E2 -16628.417} C_VEL
LIN {X 0,Y 296.575,Z 930.735,A -85,B 0,C 180,E1 -16629.733,E2 -16629.733} C_VEL
LIN {X 0,Y 294.839,Z 941.02,A -85,B 0,C 180,E1 -16631.239,E2 -16631.239} C_VEL
LIN {X 0,Y 293.393,Z 950.344,A -85,B 0,C 180,E1 -16632.947,E2 -16632.947} C_VEL
LIN {X 0,Y 292.149,Z 958.068,A -85,B 0,C 180,E1 -16634.666,E2 -16634.666} C_VEL
LIN {X 0,Y 291.142,Z 965.705,A -85,B 0,C 180,E1 -16636.753,E2 -16636.753} C_VEL
LIN {X 0,Y 290.528,Z 971.879,A -85,B 0,C 180,E1 -16638.852,E2 -16638.852} C_VEL
LIN {X 0,Y 290.301,Z 976.805,A -85,B 0,C 180,E1 -16640.956,E2 -16640.956} C_VEL
LIN {X 0,Y 290.405,Z 980.617,A -85,B 0,C 180,E1 -16643.06,E2 -16643.06} C_VEL
LIN {X 0,Y 290.495,Z 982.586,A -85,B 0,C 180,E1 -16644.456,E2 -16644.456} C_VEL
LIN {X 0,Y 290.738,Z 984.088,A -85,B 0,C 180,E1 -16645.851,E2 -16645.851} C_VEL
LIN {X 0,Y 290.831,Z 985.146,A -85,B 0,C 180,E1 -16647.239,E2 -16647.239} C_VEL
LIN {X 0,Y 290.955,Z 985.799,A -85,B 0,C 180,E1 -16648.625,E2 -16648.625} C_VEL
LIN {X 0,Y 291.081,Z 986.038,A -85,B 0,C 180,E1 -16650.009,E2 -16650.009} C_VEL
LIN {X 0,Y 290.955,Z 985.786,A -85,B 0,C 180,E1 -16651.393,E2 -16651.393} C_VEL
LIN {X 0,Y 290.831,Z 985.122,A -85,B 0,C 180,E1 -16652.779,E2 -16652.779} C_VEL
LIN {X 0,Y 290.732,Z 984.052,A -85,B 0,C 180,E1 -16654.168,E2 -16654.168} C_VEL
LIN {X 0,Y 290.474,Z 982.534,A -85,B 0,C 180,E1 -16655.563,E2 -16655.563} C_VEL
LIN {X 0,Y 290.304,Z 979.412,A -85,B 0,C 180,E1 -16657.66,E2 -16657.66} C_VEL
LIN {X 0,Y 290.683,Z 970.898,A -85,B 0,C 180,E1 -16661.868,E2 -16661.868} C_VEL
LIN {X 0,Y 291.623,Z 964.219,A -85,B 0,C 180,E1 -16664.31,E2 -16664.31} C_VEL
LIN {X 0,Y 292.687,Z 958.032,A -85,B 0,C 180,E1 -16666.161,E2 -16666.161} C_VEL
LIN {X 0,Y 294.407,Z 950.2,A -85,B 0,C 180,E1 -16668.087,E2 -16668.087} C_VEL
LIN {X 0,Y 296.296,Z 941.965,A -85,B 0,C 180,E1 -16669.763,E2 -16669.763} C_VEL
LIN {X 0,Y 298.328,Z 933.38,A -85,B 0,C 180,E1 -16671.244,E2 -16671.244} C_VEL
LIN {X 0,Y 300.77,Z 923.185,A -85,B 0,C 180,E1 -16672.686,E2 -16672.686} C_VEL
LIN {X 0,Y 302.908,Z 913.807,A -85,B 0,C 180,E1 -16673.782,E2 -16673.782} C_VEL
LIN {X 0,Y 304.937,Z 904.507,A -85,B 0,C 180,E1 -16674.699,E2 -16674.699} C_VEL
LIN {X 0,Y 307.118,Z 893.304,A -85,B 0,C 180,E1 -16675.598,E2 -16675.598} C_VEL
LIN {X 0,Y 309.019,Z 881.708,A -85,B 0,C 180,E1 -16676.334,E2 -16676.334} C_VEL
LIN {X 0,Y 310.621,Z 869.702,A -85,B 0,C 180,E1 -16676.913,E2 -16676.913} C_VEL
LIN {X 0,Y 313.812,Z 835.223,A -85,B 0,C 180,E1 -16678.298,E2 -16678.298} C_VEL
LIN {X 0,Y 314.04,Z 812.603,A -85,B 0,C 180,E1 -16679.609,E2 -16679.609} C_VEL
LIN {X 0,Y 313.374,Z 794.647,A -85,B 0,C 180,E1 -16680.924,E2 -16680.924} C_VEL
LIN {X 0,Y 312.298,Z 775.699,A -85,B 0,C 180,E1 -16682.554,E2 -16682.554} C_VEL
LIN {X 0,Y 311.283,Z 762.162,A -85,B 0,C 180,E1 -16683.92,E2 -16683.92} C_VEL
LIN {X 0,Y 309.626,Z 755.74,A -85,B 0,C 180,E1 -16685.034,E2 -16685.034} C_VEL
LIN {X 0,Y 306.314,Z 744.316,A -85,B 0,C 180,E1 -16687.537,E2 -16687.537} C_VEL
LIN {X 0,Y 304.356,Z 736.651,A -85,B 0,C 180,E1 -16689.597,E2 -16689.597} C_VEL
LIN {X 0,Y 301.768,Z 732.448,A -85,B 0,C 180,E1 -16692.493,E2 -16692.493} C_VEL
LIN {X 0,Y 300.784,Z 731.016,A -85,B 0,C 180,E1 -16694.513,E2 -16694.513} C_VEL
LIN {X 0,Y 300.634,Z 730.301,A -85,B 0,C 180,E1 -16697.317,E2 -16697.317} C_VEL
LIN {X 0,Y 301.571,Z 730.643,A -85,B 0,C 180,E1 -16699.541,E2 -16699.541} C_VEL
LIN {X 0,Y 303.801,Z 732.209,A -85,B 0,C 180,E1 -16702.082,E2 -16702.082} C_VEL
LIN {X 0,Y 305.56,Z 733.67,A -85,B 0,C 180,E1 -16703.485,E2 -16703.485} C_VEL
LIN {X 0,Y 307.364,Z 737.014,A -85,B 0,C 180,E1 -16704.894,E2 -16704.894} C_VEL
LIN {X 0,Y 308.913,Z 738.778,A -85,B 0,C 180,E1 -16705.804,E2 -16705.804} C_VEL
LIN {X 0,Y 311.385,Z 742.585,A -85,B 0,C 180,E1 -16707.169,E2 -16707.169} C_VEL
LIN {X 0,Y 314.827,Z 748.403,A -85,B 0,C 180,E1 -16708.82,E2 -16708.82} C_VEL
LIN {X 0,Y 317.8,Z 753.697,A -85,B 0,C 180,E1 -16710.078,E2 -16710.078} C_VEL
LIN {X 0,Y 320.367,Z 758.801,A -85,B 0,C 180,E1 -16711.092,E2 -16711.092} C_VEL
LIN {X 0,Y 316.274,Z 799.544,A -85,B 0,C 180,E1 -16712.793,E2 -16712.793} C_VEL
LIN {X 0,Y 315.004,Z 817.477,A -85,B 0,C 180,E1 -16713.718,E2 -16713.718} C_VEL
LIN {X 0,Y 313.781,Z 830.235,A -85,B 0,C 180,E1 -16714.602,E2 -16714.602} C_VEL
LIN {X 0,Y 312.027,Z 842.472,A -85,B 0,C 180,E1 -16715.729,E2 -16715.729} C_VEL
LIN {X 0,Y 310.425,Z 851.997,A -85,B 0,C 180,E1 -16716.836,E2 -16716.836} C_VEL
LIN {X 0,Y 308.748,Z 860.191,A -85,B 0,C 180,E1 -16717.939,E2 -16717.939} C_VEL
LIN {X 0,Y 307.064,Z 867.99,A -85,B 0,C 180,E1 -16719.221,E2 -16719.221} C_VEL
LIN {X 0,Y 305.346,Z 874.675,A -85,B 0,C 180,E1 -16720.504,E2 -16720.504} C_VEL
LIN {X 0,Y 303.357,Z 881.696,A -85,B 0,C 180,E1 -16722.124,E2 -16722.124} C_VEL
LIN {X 0,Y 301.553,Z 887.532,A -85,B 0,C 180,E1 -16723.759,E2 -16723.759} C_VEL
LIN {X 0,Y 299.514,Z 893.179,A -85,B 0,C 180,E1 -16725.737,E2 -16725.737} C_VEL
LIN {X 0,Y 297.699,Z 897.563,A -85,B 0,C 180,E1 -16727.733,E2 -16727.733} C_VEL
LIN {X 0,Y 296.67,Z 899.868,A -85,B 0,C 180,E1 -16729.075,E2 -16729.075} C_VEL
LIN {X 0,Y 295.693,Z 901.741,A -85,B 0,C 180,E1 -16730.423,E2 -16730.423} C_VEL
LIN {X 0,Y 294.789,Z 902.997,A -85,B 0,C 180,E1 -16731.776,E2 -16731.776} C_VEL
LIN {X 0,Y 293.56,Z 904.365,A -85,B 0,C 180,E1 -16734.505,E2 -16734.505} C_VEL
LIN {X 0,Y 293.097,Z 904.351,A -85,B 0,C 180,E1 -16735.875,E2 -16735.875} C_VEL
LIN {X 0,Y 292.551,Z 903.933,A -85,B 0,C 180,E1 -16737.246,E2 -16737.246} C_VEL
LIN {X 0,Y 292.274,Z 903.071,A -85,B 0,C 180,E1 -16738.622,E2 -16738.622} C_VEL
LIN {X 0,Y 291.822,Z 901.711,A -85,B 0,C 180,E1 -16740,E2 -16740} C_VEL
LIN {X 0,Y 291.61,Z 898.91,A -85,B 0,C 180,E1 -16742.072,E2 -16742.072} C_VEL
LIN {X 0,Y 291.384,Z 895.065,A -85,B 0,C 180,E1 -16744.15,E2 -16744.15} C_VEL
LIN {X 0,Y 291.791,Z 890.038,A -85,B 0,C 180,E1 -16746.222,E2 -16746.222} C_VEL
LIN {X 0,Y 292.184,Z 882.617,A -85,B 0,C 180,E1 -16748.615,E2 -16748.615} C_VEL
LIN {X 0,Y 292.549,Z 875.816,A -85,B 0,C 180,E1 -16750.379,E2 -16750.379} C_VEL
LIN {X 0,Y 293.099,Z 867.793,A -85,B 0,C 180,E1 -16752.111,E2 -16752.111} C_VEL
LIN {X 0,Y 293.677,Z 859.187,A -85,B 0,C 180,E1 -16753.67,E2 -16753.67} C_VEL
LIN {X 0,Y 294.175,Z 850.091,A -85,B 0,C 180,E1 -16755.059,E2 -16755.059} C_VEL
LIN {X 0,Y 294.878,Z 840.668,A -85,B 0,C 180,E1 -16756.263,E2 -16756.263} C_VEL
LIN {X 0,Y 295.409,Z 830.972,A -85,B 0,C 180,E1 -16757.301,E2 -16757.301} C_VEL
LIN {X 0,Y 295.909,Z 820.349,A -85,B 0,C 180,E1 -16758.232,E2 -16758.232} C_VEL
LIN {X 0,Y 296.241,Z 810.175,A -85,B 0,C 180,E1 -16758.948,E2 -16758.948} C_VEL
LIN {X 0,Y 296.51,Z 799.783,A -85,B 0,C 180,E1 -16759.515,E2 -16759.515} C_VEL
LIN {X 0,Y 296.762,Z 784.126,A -85,B 0,C 180,E1 -16760.129,E2 -16760.129} C_VEL
LIN {X 0,Y 297.977,Z 737.406,A -85,B 0,C 180,E1 -16761.72,E2 -16761.72} C_VEL
LIN {X 0,Y 291.457,Z 716.18,A -85,B 0,C 180,E1 -16762.792,E2 -16762.792} C_VEL
LIN {X 0,Y 291.376,Z 716.187,A -85,B 0,C 180,E1 -16767.276,E2 -16767.276} C_VEL
LIN {X 0,Y 291.327,Z 716.195,A -85,B 0,C 180,E1 -16770.438,E2 -16770.438} C_VEL
LIN {X 0,Y 291.366,Z 716.187,A -85,B 0,C 180,E1 -16773.696,E2 -16773.696} C_VEL
LIN {X 0,Y 291.371,Z 716.19,A -85,B 0,C 180,E1 -16777.243,E2 -16777.243} C_VEL
LIN {X 0,Y 291.322,Z 716.195,A -85,B 0,C 180,E1 -16780.645,E2 -16780.645} C_VEL
LIN {X 0,Y 291.304,Z 716.191,A -85,B 0,C 180,E1 -16784.4,E2 -16784.4} C_VEL
LIN {X 0,Y 291.315,Z 716.191,A -85,B 0,C 180,E1 -16788.407,E2 -16788.407} C_VEL
LIN {X 0,Y 291.353,Z 716.186,A -85,B 0,C 180,E1 -16791.15,E2 -16791.15} C_VEL
LIN {X 0,Y 291.375,Z 716.185,A -85,B 0,C 180,E1 -16794.62,E2 -16794.62} C_VEL
LIN {X 0,Y 291.383,Z 716.184,A -85,B 0,C 180,E1 -16797.944,E2 -16797.944} C_VEL
LIN {X 0,Y 291.384,Z 716.184,A -85,B 0,C 180,E1 -16802.482,E2 -16802.482} C_VEL
LIN {X 0,Y 291.391,Z 716.279,A -85,B 0,C 180,E1 -16802.572,E2 -16802.572} C_VEL
LIN {X 0,Y 292.461,Z 719.171,A -85,B 0,C 180,E1 -16802.765,E2 -16802.765} C_VEL
LIN {X 0,Y 300.731,Z 735.712,A -85,B 0,C 180,E1 -16804.044,E2 -16804.044} C_VEL
LIN {X 0,Y 305.487,Z 746.416,A -85,B 0,C 180,E1 -16804.772,E2 -16804.772} C_VEL
LIN {X 0,Y 304.681,Z 791.888,A -85,B 0,C 180,E1 -16805.863,E2 -16805.863} C_VEL
LIN {X 0,Y 304.526,Z 805.841,A -85,B 0,C 180,E1 -16806.318,E2 -16806.318} C_VEL
LIN {X 0,Y 304.042,Z 818.924,A -85,B 0,C 180,E1 -16807.033,E2 -16807.033} C_VEL
LIN {X 0,Y 303.189,Z 830.445,A -85,B 0,C 180,E1 -16807.9,E2 -16807.9} C_VEL
LIN {X 0,Y 302.056,Z 842.022,A -85,B 0,C 180,E1 -16809.043,E2 -16809.043} C_VEL
LIN {X 0,Y 300.723,Z 852.489,A -85,B 0,C 180,E1 -16810.362,E2 -16810.362} C_VEL
LIN {X 0,Y 299.315,Z 862.085,A -85,B 0,C 180,E1 -16811.866,E2 -16811.866} C_VEL
LIN {X 0,Y 298.02,Z 870.778,A -85,B 0,C 180,E1 -16813.553,E2 -16813.553} C_VEL
LIN {X 0,Y 296.42,Z 879.281,A -85,B 0,C 180,E1 -16815.576,E2 -16815.576} C_VEL
LIN {X 0,Y 295.067,Z 886.043,A -85,B 0,C 180,E1 -16817.613,E2 -16817.613} C_VEL
LIN {X 0,Y 294.235,Z 891.407,A -85,B 0,C 180,E1 -16819.672,E2 -16819.672} C_VEL
LIN {X 0,Y 293.697,Z 894.343,A -85,B 0,C 180,E1 -16821.043,E2 -16821.043} C_VEL
LIN {X 0,Y 292.696,Z 897.903,A -85,B 0,C 180,E1 -16823.096,E2 -16823.096} C_VEL
LIN {X 0,Y 292.295,Z 899.725,A -85,B 0,C 180,E1 -16824.472,E2 -16824.472} C_VEL
LIN {X 0,Y 292.041,Z 902.036,A -85,B 0,C 180,E1 -16827.232,E2 -16827.232} C_VEL
LIN {X 0,Y 291.803,Z 902.877,A -85,B 0,C 180,E1 -16829.991,E2 -16829.991} C_VEL
LIN {X 0,Y 292.039,Z 902.113,A -85,B 0,C 180,E1 -16832.749,E2 -16832.749} C_VEL
LIN {X 0,Y 292.276,Z 899.882,A -85,B 0,C 180,E1 -16835.51,E2 -16835.51} C_VEL
LIN {X 0,Y 292.955,Z 897.064,A -85,B 0,C 180,E1 -16837.572,E2 -16837.572} C_VEL
LIN {X 0,Y 293.888,Z 893.236,A -85,B 0,C 180,E1 -16839.627,E2 -16839.627} C_VEL
LIN {X 0,Y 294.843,Z 887.764,A -85,B 0,C 180,E1 -16841.896,E2 -16841.896} C_VEL
LIN {X 0,Y 296.148,Z 880.95,A -85,B 0,C 180,E1 -16844.068,E2 -16844.068} C_VEL
LIN {X 0,Y 297.685,Z 872.92,A -85,B 0,C 180,E1 -16846.095,E2 -16846.095} C_VEL
LIN {X 0,Y 299.028,Z 864.7,A -85,B 0,C 180,E1 -16847.78,E2 -16847.78} C_VEL
LIN {X 0,Y 300.476,Z 854.528,A -85,B 0,C 180,E1 -16849.458,E2 -16849.458} C_VEL
LIN {X 0,Y 301.907,Z 844.057,A -85,B 0,C 180,E1 -16850.829,E2 -16850.829} C_VEL
LIN {X 0,Y 303.105,Z 832.786,A -85,B 0,C 180,E1 -16852.002,E2 -16852.002} C_VEL
LIN {X 0,Y 304.077,Z 820.856,A -85,B 0,C 180,E1 -16852.945,E2 -16852.945} C_VEL
LIN {X 0,Y 304.52,Z 808.928,A -85,B 0,C 180,E1 -16853.646,E2 -16853.646} C_VEL
LIN {X 0,Y 304.719,Z 797.05,A -85,B 0,C 180,E1 -16854.109,E2 -16854.109} C_VEL
LIN {X 0,Y 305.389,Z 755.621,A -85,B 0,C 180,E1 -16855.119,E2 -16855.119} C_VEL
LIN {X 0,Y 305.568,Z 746.583,A -85,B 0,C 180,E1 -16855.335,E2 -16855.335} C_VEL
LIN {X 0,Y 297.04,Z 727.852,A -85,B 0,C 180,E1 -16856.65,E2 -16856.65} C_VEL
LIN {X 0,Y 291.559,Z 716.972,A -85,B 0,C 180,E1 -16857.514,E2 -16857.514} C_VEL
LIN {X 0,Y 291.409,Z 716.179,A -85,B 0,C 180,E1 -16857.586,E2 -16857.586} C_VEL
LIN {X 0,Y 291.307,Z 716.195,A -85,B 0,C 180,E1 -16860.427,E2 -16860.427} C_VEL
LIN {X 0,Y 291.313,Z 716.196,A -85,B 0,C 180,E1 -16863.689,E2 -16863.689} C_VEL
LIN {X 0,Y 291.363,Z 716.179,A -85,B 0,C 180,E1 -16867.25,E2 -16867.25} C_VEL
LIN {X 0,Y 291.363,Z 716.193,A -85,B 0,C 180,E1 -16870.622,E2 -16870.622} C_VEL
LIN {X 0,Y 291.364,Z 716.17,A -85,B 0,C 180,E1 -16874.371,E2 -16874.371} C_VEL
LIN {X 0,Y 291.345,Z 716.19,A -85,B 0,C 180,E1 -16877.757,E2 -16877.757} C_VEL
LIN {X 0,Y 290.662,Z 716.283,A -85,B 0,C 180,E1 -16878.911,E2 -16878.911} C_VEL
LIN {X 0,Y 287.815,Z 716.644,A -85,B 0,C 180,E1 -16880.79,E2 -16880.79} C_VEL
LIN {X 0,Y 285.41,Z 716.942,A -85,B 0,C 180,E1 -16882.316,E2 -16882.316} C_VEL
LIN {X 0,Y 284.379,Z 717.063,A -85,B 0,C 180,E1 -16883.498,E2 -16883.498} C_VEL
LIN {X 0,Y 284.295,Z 717.071,A -85,B 0,C 180,E1 -16883.898,E2 -16883.898} C_VEL
LIN {X 0,Y 284.256,Z 717.072,A -85,B 0,C 180,E1 -16887.182,E2 -16887.182} C_VEL
LIN {X 0,Y 284.303,Z 717.06,A -85,B 0,C 180,E1 -16890.369,E2 -16890.369} C_VEL
LIN {X 0,Y 284.318,Z 717.067,A -85,B 0,C 180,E1 -16893.58,E2 -16893.58} C_VEL
LIN {X 0,Y 284.276,Z 717.063,A -85,B 0,C 180,E1 -16896.699,E2 -16896.699} C_VEL
LIN {X 0,Y 284.34,Z 717.058,A -85,B 0,C 180,E1 -16901.257,E2 -16901.257} C_VEL
LIN {X 0,Y 284.415,Z 717.052,A -85,B 0,C 180,E1 -16904.466,E2 -16904.466} C_VEL
LIN {X 0,Y 284.423,Z 717.045,A -85,B 0,C 180,E1 -16908.599,E2 -16908.599} C_VEL
LIN {X 0,Y 284.587,Z 717.036,A -85,B 0,C 180,E1 -16911.479,E2 -16911.479} C_VEL
LIN {X 0,Y 284.535,Z 717.043,A -85,B 0,C 180,E1 -16914.33,E2 -16914.33} C_VEL
LIN {X 0,Y 284.794,Z 717.011,A -85,B 0,C 180,E1 -16918.586,E2 -16918.586} C_VEL
LIN {X 0,Y 284.794,Z 717.005,A -85,B 0,C 180,E1 -16921.414,E2 -16921.414} C_VEL
LIN {X 0,Y 284.535,Z 717.046,A -85,B 0,C 180,E1 -16925.67,E2 -16925.67} C_VEL
LIN {X 0,Y 284.597,Z 717.024,A -85,B 0,C 180,E1 -16929.05,E2 -16929.05} C_VEL
LIN {X 0,Y 284.411,Z 717.059,A -85,B 0,C 180,E1 -16932.85,E2 -16932.85} C_VEL
LIN {X 0,Y 284.419,Z 717.056,A -85,B 0,C 180,E1 -16935.772,E2 -16935.772} C_VEL
LIN {X 0,Y 284.316,Z 717.057,A -85,B 0,C 180,E1 -16940.247,E2 -16940.247} C_VEL
LIN {X 0,Y 284.307,Z 717.069,A -85,B 0,C 180,E1 -16943.879,E2 -16943.879} C_VEL
LIN {X 0,Y 284.338,Z 717.06,A -85,B 0,C 180,E1 -16947.178,E2 -16947.178} C_VEL
LIN {X 0,Y 284.243,Z 717.072,A -85,B 0,C 180,E1 -16951.281,E2 -16951.281} C_VEL
LIN {X 0,Y 284.31,Z 717.068,A -85,B 0,C 180,E1 -16955.361,E2 -16955.361} C_VEL
LIN {X 0,Y 284.282,Z 717.054,A -85,B 0,C 180,E1 -16958.174,E2 -16958.174} C_VEL
LIN {X 0,Y 284.297,Z 717.071,A -85,B 0,C 180,E1 -16962.149,E2 -16962.149} C_VEL
LIN {X 0,Y 284.312,Z 717.069,A -85,B 0,C 180,E1 -16966.217,E2 -16966.217} C_VEL
LIN {X 0,Y 284.351,Z 717.238,A -85,B 0,C 180,E1 -16968.466,E2 -16968.466} C_VEL
LIN {X 0,Y 287.117,Z 727.543,A -85,B 0,C 180,E1 -16971.563,E2 -16971.563} C_VEL
LIN {X 0,Y 289.833,Z 738.745,A -85,B 0,C 180,E1 -16974.712,E2 -16974.712} C_VEL
LIN {X 0,Y 292.528,Z 751.591,A -85,B 0,C 180,E1 -16978.106,E2 -16978.106} C_VEL
LIN {X 0,Y 290.08,Z 767.595,A -85,B 0,C 180,E1 -16981.756,E2 -16981.756} C_VEL
LIN {X 0,Y 293.735,Z 796.76,A -85,B 0,C 180,E1 -16982.904,E2 -16982.904} C_VEL
LIN {X 0,Y 296.723,Z 827.475,A -85,B 0,C 180,E1 -16983.993,E2 -16983.993} C_VEL
LIN {X 0,Y 297.26,Z 835.148,A -85,B 0,C 180,E1 -16984.241,E2 -16984.241} C_VEL
LIN {X 0,Y 295.946,Z 879.334,A -85,B 0,C 180,E1 -16985.32,E2 -16985.32} C_VEL
LIN {X 0,Y 294.959,Z 893.132,A -85,B 0,C 180,E1 -16985.931,E2 -16985.931} C_VEL
LIN {X 0,Y 293.597,Z 905.595,A -85,B 0,C 180,E1 -16986.748,E2 -16986.748} C_VEL
LIN {X 0,Y 291.783,Z 918.358,A -85,B 0,C 180,E1 -16987.904,E2 -16987.904} C_VEL
LIN {X 0,Y 289.918,Z 929.725,A -85,B 0,C 180,E1 -16989.247,E2 -16989.247} C_VEL
LIN {X 0,Y 288.13,Z 940.011,A -85,B 0,C 180,E1 -16990.786,E2 -16990.786} C_VEL
LIN {X 0,Y 286.55,Z 949.324,A -85,B 0,C 180,E1 -16992.527,E2 -16992.527} C_VEL
LIN {X 0,Y 285.16,Z 957.035,A -85,B 0,C 180,E1 -16994.281,E2 -16994.281} C_VEL
LIN {X 0,Y 284.477,Z 962.334,A -85,B 0,C 180,E1 -16995.708,E2 -16995.708} C_VEL
LIN {X 0,Y 283.69,Z 968.971,A -85,B 0,C 180,E1 -16997.854,E2 -16997.854} C_VEL
LIN {X 0,Y 283.279,Z 974.283,A -85,B 0,C 180,E1 -17000.009,E2 -17000.009} C_VEL
LIN {X 0,Y 283.253,Z 978.459,A -85,B 0,C 180,E1 -17002.167,E2 -17002.167} C_VEL
LIN {X 0,Y 283.417,Z 981.572,A -85,B 0,C 180,E1 -17004.317,E2 -17004.317} C_VEL
LIN {X 0,Y 283.656,Z 983.075,A -85,B 0,C 180,E1 -17005.747,E2 -17005.747} C_VEL
LIN {X 0,Y 283.781,Z 984.139,A -85,B 0,C 180,E1 -17007.171,E2 -17007.171} C_VEL
LIN {X 0,Y 283.914,Z 984.795,A -85,B 0,C 180,E1 -17008.591,E2 -17008.591} C_VEL
LIN {X 0,Y 284.048,Z 985.034,A -85,B 0,C 180,E1 -17010.009,E2 -17010.009} C_VEL
LIN {X 0,Y 283.914,Z 984.78,A -85,B 0,C 180,E1 -17011.428,E2 -17011.428} C_VEL
LIN {X 0,Y 283.78,Z 984.115,A -85,B 0,C 180,E1 -17012.848,E2 -17012.848} C_VEL
LIN {X 0,Y 283.649,Z 983.039,A -85,B 0,C 180,E1 -17014.272,E2 -17014.272} C_VEL
LIN {X 0,Y 283.392,Z 981.518,A -85,B 0,C 180,E1 -17015.702,E2 -17015.702} C_VEL
LIN {X 0,Y 283.245,Z 978.394,A -85,B 0,C 180,E1 -17017.852,E2 -17017.852} C_VEL
LIN {X 0,Y 283.46,Z 971.779,A -85,B 0,C 180,E1 -17021.449,E2 -17021.449} C_VEL
LIN {X 0,Y 284.188,Z 966.794,A -85,B 0,C 180,E1 -17023.597,E2 -17023.597} C_VEL
LIN {X 0,Y 285.053,Z 961.765,A -85,B 0,C 180,E1 -17025.378,E2 -17025.378} C_VEL
LIN {X 0,Y 286.449,Z 955.823,A -85,B 0,C 180,E1 -17027.131,E2 -17027.131} C_VEL
LIN {X 0,Y 288,Z 948.908,A -85,B 0,C 180,E1 -17028.873,E2 -17028.873} C_VEL
LIN {X 0,Y 290.12,Z 940.784,A -85,B 0,C 180,E1 -17030.572,E2 -17030.572} C_VEL
LIN {X 0,Y 292.337,Z 932.189,A -85,B 0,C 180,E1 -17032.072,E2 -17032.072} C_VEL
LIN {X 0,Y 294.928,Z 922.161,A -85,B 0,C 180,E1 -17033.533,E2 -17033.533} C_VEL
LIN {X 0,Y 297.222,Z 912.991,A -85,B 0,C 180,E1 -17034.638,E2 -17034.638} C_VEL
LIN {X 0,Y 299.715,Z 902.059,A -85,B 0,C 180,E1 -17035.717,E2 -17035.717} C_VEL
LIN {X 0,Y 302.052,Z 890.82,A -85,B 0,C 180,E1 -17036.617,E2 -17036.617} C_VEL
LIN {X 0,Y 304.065,Z 879.26,A -85,B 0,C 180,E1 -17037.355,E2 -17037.355} C_VEL
LIN {X 0,Y 305.778,Z 867.306,A -85,B 0,C 180,E1 -17037.932,E2 -17037.932} C_VEL
LIN {X 0,Y 308.848,Z 836.235,A -85,B 0,C 180,E1 -17039.218,E2 -17039.218} C_VEL
LIN {X 0,Y 309.33,Z 814.647,A -85,B 0,C 180,E1 -17040.51,E2 -17040.51} C_VEL
LIN {X 0,Y 308.961,Z 797.514,A -85,B 0,C 180,E1 -17041.807,E2 -17041.807} C_VEL
LIN {X 0,Y 308.256,Z 778.904,A -85,B 0,C 180,E1 -17043.455,E2 -17043.455} C_VEL
LIN {X 0,Y 307.556,Z 765.899,A -85,B 0,C 180,E1 -17044.817,E2 -17044.817} C_VEL
LIN {X 0,Y 306.249,Z 760.357,A -85,B 0,C 180,E1 -17045.82,E2 -17045.82} C_VEL
LIN {X 0,Y 303.372,Z 749.216,A -85,B 0,C 180,E1 -17048.355,E2 -17048.355} C_VEL
LIN {X 0,Y 302.022,Z 742.838,A -85,B 0,C 180,E1 -17050.11,E2 -17050.11} C_VEL
LIN {X 0,Y 299.838,Z 739.073,A -85,B 0,C 180,E1 -17052.832,E2 -17052.832} C_VEL
LIN {X 0,Y 298.925,Z 737.652,A -85,B 0,C 180,E1 -17055.144,E2 -17055.144} C_VEL
LIN {X 0,Y 298.897,Z 737.215,A -85,B 0,C 180,E1 -17057.009,E2 -17057.009} C_VEL
LIN {X 0,Y 299.774,Z 737.455,A -85,B 0,C 180,E1 -17059.397,E2 -17059.397} C_VEL
LIN {X 0,Y 301.903,Z 739.017,A -85,B 0,C 180,E1 -17061.945,E2 -17061.945} C_VEL
LIN {X 0,Y 303.376,Z 740.34,A -85,B 0,C 180,E1 -17063.189,E2 -17063.189} C_VEL
LIN {X 0,Y 305.151,Z 743.602,A -85,B 0,C 180,E1 -17064.644,E2 -17064.644} C_VEL
LIN {X 0,Y 306.289,Z 744.991,A -85,B 0,C 180,E1 -17065.376,E2 -17065.376} C_VEL
LIN {X 0,Y 309.407,Z 750.22,A -85,B 0,C 180,E1 -17067.196,E2 -17067.196} C_VEL
LIN {X 0,Y 312.728,Z 755.964,A -85,B 0,C 180,E1 -17068.815,E2 -17068.815} C_VEL
LIN {X 0,Y 315.877,Z 762.298,A -85,B 0,C 180,E1 -17070.204,E2 -17070.204} C_VEL
LIN {X 0,Y 311.749,Z 798.471,A -85,B 0,C 180,E1 -17071.743,E2 -17071.743} C_VEL
LIN {X 0,Y 310.273,Z 817.398,A -85,B 0,C 180,E1 -17072.711,E2 -17072.711} C_VEL
LIN {X 0,Y 309.167,Z 828.114,A -85,B 0,C 180,E1 -17073.445,E2 -17073.445} C_VEL
LIN {X 0,Y 307.567,Z 839.732,A -85,B 0,C 180,E1 -17074.45,E2 -17074.45} C_VEL
LIN {X 0,Y 305.57,Z 851.453,A -85,B 0,C 180,E1 -17075.725,E2 -17075.725} C_VEL
LIN {X 0,Y 303.514,Z 860.857,A -85,B 0,C 180,E1 -17076.999,E2 -17076.999} C_VEL
LIN {X 0,Y 301.418,Z 869.544,A -85,B 0,C 180,E1 -17078.455,E2 -17078.455} C_VEL
LIN {X 0,Y 299.439,Z 876.734,A -85,B 0,C 180,E1 -17079.869,E2 -17079.869} C_VEL
LIN {X 0,Y 297.574,Z 882.883,A -85,B 0,C 180,E1 -17081.322,E2 -17081.322} C_VEL
LIN {X 0,Y 295.488,Z 888.93,A -85,B 0,C 180,E1 -17083.061,E2 -17083.061} C_VEL
LIN {X 0,Y 293.682,Z 893.724,A -85,B 0,C 180,E1 -17084.738,E2 -17084.738} C_VEL
LIN {X 0,Y 292.34,Z 896.986,A -85,B 0,C 180,E1 -17086.09,E2 -17086.09} C_VEL
LIN {X 0,Y 290.549,Z 900.722,A -85,B 0,C 180,E1 -17088.135,E2 -17088.135} C_VEL
LIN {X 0,Y 288.89,Z 903.387,A -85,B 0,C 180,E1 -17090.195,E2 -17090.195} C_VEL
LIN {X 0,Y 287.943,Z 904.586,A -85,B 0,C 180,E1 -17091.579,E2 -17091.579} C_VEL
LIN {X 0,Y 286.624,Z 905.679,A -85,B 0,C 180,E1 -17094.371,E2 -17094.371} C_VEL
LIN {X 0,Y 286.134,Z 905.546,A -85,B 0,C 180,E1 -17095.774,E2 -17095.774} C_VEL
LIN {X 0,Y 285.551,Z 905.03,A -85,B 0,C 180,E1 -17097.179,E2 -17097.179} C_VEL
LIN {X 0,Y 285.262,Z 904.014,A -85,B 0,C 180,E1 -17098.588,E2 -17098.588} C_VEL
LIN {X 0,Y 284.793,Z 902.583,A -85,B 0,C 180,E1 -17100,E2 -17100} C_VEL
LIN {X 0,Y 284.552,Z 899.601,A -85,B 0,C 180,E1 -17102.123,E2 -17102.123} C_VEL
LIN {X 0,Y 284.346,Z 895.567,A -85,B 0,C 180,E1 -17104.252,E2 -17104.252} C_VEL
LIN {X 0,Y 284.802,Z 889.288,A -85,B 0,C 180,E1 -17106.731,E2 -17106.731} C_VEL
LIN {X 0,Y 285.085,Z 883.732,A -85,B 0,C 180,E1 -17108.506,E2 -17108.506} C_VEL
LIN {X 0,Y 285.462,Z 877.075,A -85,B 0,C 180,E1 -17110.282,E2 -17110.282} C_VEL
LIN {X 0,Y 285.996,Z 869.058,A -85,B 0,C 180,E1 -17112.057,E2 -17112.057} C_VEL
LIN {X 0,Y 286.593,Z 860.458,A -85,B 0,C 180,E1 -17113.652,E2 -17113.652} C_VEL
LIN {X 0,Y 287.096,Z 851.374,A -85,B 0,C 180,E1 -17115.076,E2 -17115.076} C_VEL
LIN {X 0,Y 287.777,Z 841.967,A -85,B 0,C 180,E1 -17116.311,E2 -17116.311} C_VEL
LIN {X 0,Y 288.298,Z 832.573,A -85,B 0,C 180,E1 -17117.348,E2 -17117.348} C_VEL
LIN {X 0,Y 288.834,Z 821.259,A -85,B 0,C 180,E1 -17118.367,E2 -17118.367} C_VEL
LIN {X 0,Y 289.217,Z 810.263,A -85,B 0,C 180,E1 -17119.151,E2 -17119.151} C_VEL
LIN {X 0,Y 289.519,Z 798.658,A -85,B 0,C 180,E1 -17119.775,E2 -17119.775} C_VEL
LIN {X 0,Y 290.583,Z 754.206,A -85,B 0,C 180,E1 -17121.401,E2 -17121.401} C_VEL
LIN {X 0,Y 291.031,Z 738.799,A -85,B 0,C 180,E1 -17121.951,E2 -17121.951} C_VEL
LIN {X 0,Y 284.403,Z 717.06,A -85,B 0,C 180,E1 -17123.071,E2 -17123.071} C_VEL
LIN {X 0,Y 284.353,Z 717.063,A -85,B 0,C 180,E1 -17127.143,E2 -17127.143} C_VEL
LIN {X 0,Y 284.302,Z 717.071,A -85,B 0,C 180,E1 -17131.274,E2 -17131.274} C_VEL
LIN {X 0,Y 284.36,Z 717.061,A -85,B 0,C 180,E1 -17135.343,E2 -17135.343} C_VEL
LIN {X 0,Y 284.317,Z 717.066,A -85,B 0,C 180,E1 -17138.169,E2 -17138.169} C_VEL
LIN {X 0,Y 284.258,Z 717.07,A -85,B 0,C 180,E1 -17142.112,E2 -17142.112} C_VEL
LIN {X 0,Y 284.259,Z 717.069,A -85,B 0,C 180,E1 -17146.181,E2 -17146.181} C_VEL
LIN {X 0,Y 284.305,Z 717.064,A -85,B 0,C 180,E1 -17150.025,E2 -17150.025} C_VEL
LIN {X 0,Y 284.337,Z 717.06,A -85,B 0,C 180,E1 -17153.606,E2 -17153.606} C_VEL
LIN {X 0,Y 284.325,Z 717.062,A -85,B 0,C 180,E1 -17157.185,E2 -17157.185} C_VEL
LIN {X 0,Y 284.332,Z 717.063,A -85,B 0,C 180,E1 -17161.78,E2 -17161.78} C_VEL
LIN {X 0,Y 285.529,Z 720.179,A -85,B 0,C 180,E1 -17162.043,E2 -17162.043} C_VEL
LIN {X 0,Y 294.166,Z 737.292,A -85,B 0,C 180,E1 -17163.433,E2 -17163.433} C_VEL
LIN {X 0,Y 299.083,Z 748.322,A -85,B 0,C 180,E1 -17164.216,E2 -17164.216} C_VEL
LIN {X 0,Y 298.27,Z 792.463,A -85,B 0,C 180,E1 -17165.298,E2 -17165.298} C_VEL
LIN {X 0,Y 298.103,Z 806.368,A -85,B 0,C 180,E1 -17165.753,E2 -17165.753} C_VEL
LIN {X 0,Y 297.637,Z 818.653,A -85,B 0,C 180,E1 -17166.418,E2 -17166.418} C_VEL
LIN {X 0,Y 296.689,Z 831.454,A -85,B 0,C 180,E1 -17167.389,E2 -17167.389} C_VEL
LIN {X 0,Y 295.504,Z 843.03,A -85,B 0,C 180,E1 -17168.556,E2 -17168.556} C_VEL
LIN {X 0,Y 294.113,Z 853.495,A -85,B 0,C 180,E1 -17169.902,E2 -17169.902} C_VEL
LIN {X 0,Y 292.645,Z 863.091,A -85,B 0,C 180,E1 -17171.437,E2 -17171.437} C_VEL
LIN {X 0,Y 291.287,Z 871.784,A -85,B 0,C 180,E1 -17173.162,E2 -17173.162} C_VEL
LIN {X 0,Y 289.619,Z 880.286,A -85,B 0,C 180,E1 -17175.23,E2 -17175.23} C_VEL
LIN {X 0,Y 288.206,Z 887.047,A -85,B 0,C 180,E1 -17177.314,E2 -17177.314} C_VEL
LIN {X 0,Y 287.323,Z 892.411,A -85,B 0,C 180,E1 -17179.42,E2 -17179.42} C_VEL
LIN {X 0,Y 286.757,Z 895.347,A -85,B 0,C 180,E1 -17180.825,E2 -17180.825} C_VEL
LIN {X 0,Y 285.721,Z 898.906,A -85,B 0,C 180,E1 -17182.927,E2 -17182.927} C_VEL
LIN {X 0,Y 285.3,Z 900.729,A -85,B 0,C 180,E1 -17184.336,E2 -17184.336} C_VEL
LIN {X 0,Y 285.022,Z 903.039,A -85,B 0,C 180,E1 -17187.164,E2 -17187.164} C_VEL
LIN {X 0,Y 284.776,Z 903.88,A -85,B 0,C 180,E1 -17189.991,E2 -17189.991} C_VEL
LIN {X 0,Y 285.019,Z 903.115,A -85,B 0,C 180,E1 -17192.817,E2 -17192.817} C_VEL
LIN {X 0,Y 285.281,Z 900.884,A -85,B 0,C 180,E1 -17195.645,E2 -17195.645} C_VEL
LIN {X 0,Y 285.991,Z 898.066,A -85,B 0,C 180,E1 -17197.758,E2 -17197.758} C_VEL
LIN {X 0,Y 286.962,Z 894.238,A -85,B 0,C 180,E1 -17199.861,E2 -17199.861} C_VEL
LIN {X 0,Y 287.97,Z 888.764,A -85,B 0,C 180,E1 -17202.184,E2 -17202.184} C_VEL
LIN {X 0,Y 289.336,Z 881.951,A -85,B 0,C 180,E1 -17204.406,E2 -17204.406} C_VEL
LIN {X 0,Y 290.939,Z 873.92,A -85,B 0,C 180,E1 -17206.479,E2 -17206.479} C_VEL
LIN {X 0,Y 292.343,Z 865.7,A -85,B 0,C 180,E1 -17208.2,E2 -17208.2} C_VEL
LIN {X 0,Y 293.858,Z 855.527,A -85,B 0,C 180,E1 -17209.915,E2 -17209.915} C_VEL
LIN {X 0,Y 295.349,Z 845.055,A -85,B 0,C 180,E1 -17211.313,E2 -17211.313} C_VEL
LIN {X 0,Y 296.601,Z 833.782,A -85,B 0,C 180,E1 -17212.511,E2 -17212.511} C_VEL
LIN {X 0,Y 297.614,Z 821.85,A -85,B 0,C 180,E1 -17213.472,E2 -17213.472} C_VEL
LIN {X 0,Y 298.105,Z 809.382,A -85,B 0,C 180,E1 -17214.215,E2 -17214.215} C_VEL
LIN {X 0,Y 298.31,Z 797.495,A -85,B 0,C 180,E1 -17214.678,E2 -17214.678} C_VEL
LIN {X 0,Y 299.036,Z 755.306,A -85,B 0,C 180,E1 -17215.725,E2 -17215.725} C_VEL
LIN {X 0,Y 299.054,Z 748.125,A -85,B 0,C 180,E1 -17215.913,E2 -17215.913} C_VEL
LIN {X 0,Y 290.247,Z 729.133,A -85,B 0,C 180,E1 -17217.319,E2 -17217.319} C_VEL
LIN {X 0,Y 284.625,Z 718.37,A -85,B 0,C 180,E1 -17218.235,E2 -17218.235} C_VEL
LIN {X 0,Y 284.346,Z 717.06,A -85,B 0,C 180,E1 -17218.34,E2 -17218.34} C_VEL
LIN {X 0,Y 284.276,Z 717.075,A -85,B 0,C 180,E1 -17222.935,E2 -17222.935} C_VEL
LIN {X 0,Y 284.318,Z 717.069,A -85,B 0,C 180,E1 -17226.373,E2 -17226.373} C_VEL
LIN {X 0,Y 284.315,Z 717.063,A -85,B 0,C 180,E1 -17229.978,E2 -17229.978} C_VEL
LIN {X 0,Y 284.314,Z 717.049,A -85,B 0,C 180,E1 -17234.204,E2 -17234.204} C_VEL
LIN {X 0,Y 284.296,Z 717.074,A -85,B 0,C 180,E1 -17238.128,E2 -17238.128} C_VEL
LIN {X 0,Y 284.291,Z 717.071,A -85,B 0,C 180,E1 -17242.266,E2 -17242.266} C_VEL
LIN {X 0,Y 284.295,Z 717.071,A -85,B 0,C 180,E1 -17243.898,E2 -17243.898} C_VEL
LIN {X 0,Y 283.621,Z 717.151,A -85,B 0,C 180,E1 -17245.08,E2 -17245.08} C_VEL
LIN {X 0,Y 280.75,Z 717.509,A -85,B 0,C 180,E1 -17247.005,E2 -17247.005} C_VEL
LIN {X 0,Y 278.314,Z 717.815,A -85,B 0,C 180,E1 -17248.569,E2 -17248.569} C_VEL
LIN {X 0,Y 277.268,Z 717.941,A -85,B 0,C 180,E1 -17249.781,E2 -17249.781} C_VEL
LIN {X 0,Y 277.182,Z 717.948,A -85,B 0,C 180,E1 -17250.192,E2 -17250.192} C_VEL
LIN {X 0,Y 277.301,Z 717.941,A -85,B 0,C 180,E1 -17252.858,E2 -17252.858} C_VEL
LIN {X 0,Y 277.239,Z 717.94,A -85,B 0,C 180,E1 -17256.071,E2 -17256.071} C_VEL
LIN {X 0,Y 277.283,Z 717.94,A -85,B 0,C 180,E1 -17260.762,E2 -17260.762} C_VEL
LIN {X 0,Y 277.364,Z 717.935,A -85,B 0,C 180,E1 -17265.322,E2 -17265.322} C_VEL
LIN {X 0,Y 277.442,Z 717.912,A -85,B 0,C 180,E1 -17269.786,E2 -17269.786} C_VEL
LIN {X 0,Y 277.581,Z 717.914,A -85,B 0,C 180,E1 -17272.727,E2 -17272.727} C_VEL
LIN {X 0,Y 277.76,Z 717.887,A -85,B 0,C 180,E1 -17278.55,E2 -17278.55} C_VEL
LIN {X 0,Y 277.76,Z 717.881,A -85,B 0,C 180,E1 -17281.45,E2 -17281.45} C_VEL
LIN {X 0,Y 277.506,Z 717.921,A -85,B 0,C 180,E1 -17285.814,E2 -17285.814} C_VEL
LIN {X 0,Y 277.562,Z 717.9,A -85,B 0,C 180,E1 -17289.155,E2 -17289.155} C_VEL
LIN {X 0,Y 277.351,Z 717.938,A -85,B 0,C 180,E1 -17293.183,E2 -17293.183} C_VEL
LIN {X 0,Y 277.337,Z 717.935,A -85,B 0,C 180,E1 -17296.186,E2 -17296.186} C_VEL
LIN {X 0,Y 277.284,Z 717.933,A -85,B 0,C 180,E1 -17300.354,E2 -17300.354} C_VEL
LIN {X 0,Y 277.257,Z 717.945,A -85,B 0,C 180,E1 -17304.174,E2 -17304.174} C_VEL
LIN {X 0,Y 277.267,Z 717.943,A -85,B 0,C 180,E1 -17307.51,E2 -17307.51} C_VEL
LIN {X 0,Y 277.218,Z 717.944,A -85,B 0,C 180,E1 -17310.488,E2 -17310.488} C_VEL
LIN {X 0,Y 277.202,Z 717.949,A -85,B 0,C 180,E1 -17313.902,E2 -17313.902} C_VEL
LIN {X 0,Y 277.236,Z 717.939,A -85,B 0,C 180,E1 -17317.474,E2 -17317.474} C_VEL
LIN {X 0,Y 277.248,Z 717.951,A -85,B 0,C 180,E1 -17321.23,E2 -17321.23} C_VEL
LIN {X 0,Y 277.246,Z 717.949,A -85,B 0,C 180,E1 -17325.217,E2 -17325.217} C_VEL
LIN {X 0,Y 277.271,Z 718.016,A -85,B 0,C 180,E1 -17327.709,E2 -17327.709} C_VEL
LIN {X 0,Y 280.31,Z 729.229,A -85,B 0,C 180,E1 -17331.201,E2 -17331.201} C_VEL
LIN {X 0,Y 282.875,Z 739.839,A -85,B 0,C 180,E1 -17334.277,E2 -17334.277} C_VEL
LIN {X 0,Y 285.459,Z 752.152,A -85,B 0,C 180,E1 -17337.637,E2 -17337.637} C_VEL
LIN {X 0,Y 285.589,Z 753.851,A -85,B 0,C 180,E1 -17338.07,E2 -17338.07} C_VEL
LIN {X 0,Y 283.484,Z 766.511,A -85,B 0,C 180,E1 -17341.03,E2 -17341.03} C_VEL
LIN {X 0,Y 287.302,Z 796.73,A -85,B 0,C 180,E1 -17342.273,E2 -17342.273} C_VEL
LIN {X 0,Y 290.34,Z 828.693,A -85,B 0,C 180,E1 -17343.436,E2 -17343.436} C_VEL
LIN {X 0,Y 290.758,Z 836.49,A -85,B 0,C 180,E1 -17343.684,E2 -17343.684} C_VEL
LIN {X 0,Y 289.498,Z 877.979,A -85,B 0,C 180,E1 -17344.718,E2 -17344.718} C_VEL
LIN {X 0,Y 288.518,Z 891.495,A -85,B 0,C 180,E1 -17345.319,E2 -17345.319} C_VEL
LIN {X 0,Y 287.103,Z 904.591,A -85,B 0,C 180,E1 -17346.189,E2 -17346.189} C_VEL
LIN {X 0,Y 285.465,Z 915.754,A -85,B 0,C 180,E1 -17347.197,E2 -17347.197} C_VEL
LIN {X 0,Y 283.495,Z 927.408,A -85,B 0,C 180,E1 -17348.563,E2 -17348.563} C_VEL
LIN {X 0,Y 281.566,Z 937.937,A -85,B 0,C 180,E1 -17350.129,E2 -17350.129} C_VEL
LIN {X 0,Y 279.958,Z 946.588,A -85,B 0,C 180,E1 -17351.723,E2 -17351.723} C_VEL
LIN {X 0,Y 278.569,Z 954.567,A -85,B 0,C 180,E1 -17353.511,E2 -17353.511} C_VEL
LIN {X 0,Y 277.346,Z 962.505,A -85,B 0,C 180,E1 -17355.707,E2 -17355.707} C_VEL
LIN {X 0,Y 276.469,Z 969.836,A -85,B 0,C 180,E1 -17358.277,E2 -17358.277} C_VEL
LIN {X 0,Y 276.161,Z 974.764,A -85,B 0,C 180,E1 -17360.489,E2 -17360.489} C_VEL
LIN {X 0,Y 276.234,Z 978.826,A -85,B 0,C 180,E1 -17362.861,E2 -17362.861} C_VEL
LIN {X 0,Y 276.334,Z 980.557,A -85,B 0,C 180,E1 -17364.171,E2 -17364.171} C_VEL
LIN {X 0,Y 276.578,Z 982.063,A -85,B 0,C 180,E1 -17365.638,E2 -17365.638} C_VEL
LIN {X 0,Y 276.727,Z 983.132,A -85,B 0,C 180,E1 -17367.098,E2 -17367.098} C_VEL
LIN {X 0,Y 276.872,Z 983.79,A -85,B 0,C 180,E1 -17368.555,E2 -17368.555} C_VEL
LIN {X 0,Y 277.016,Z 984.031,A -85,B 0,C 180,E1 -17370.01,E2 -17370.01} C_VEL
LIN {X 0,Y 276.871,Z 983.775,A -85,B 0,C 180,E1 -17371.464,E2 -17371.464} C_VEL
LIN {X 0,Y 276.726,Z 983.107,A -85,B 0,C 180,E1 -17372.921,E2 -17372.921} C_VEL
LIN {X 0,Y 276.569,Z 982.025,A -85,B 0,C 180,E1 -17374.382,E2 -17374.382} C_VEL
LIN {X 0,Y 276.213,Z 978.841,A -85,B 0,C 180,E1 -17377.104,E2 -17377.104} C_VEL
LIN {X 0,Y 276.293,Z 972.636,A -85,B 0,C 180,E1 -17381.007,E2 -17381.007} C_VEL
LIN {X 0,Y 276.935,Z 968.205,A -85,B 0,C 180,E1 -17383.212,E2 -17383.212} C_VEL
LIN {X 0,Y 278.132,Z 961.579,A -85,B 0,C 180,E1 -17385.771,E2 -17385.771} C_VEL
LIN {X 0,Y 279.968,Z 954.607,A -85,B 0,C 180,E1 -17387.918,E2 -17387.918} C_VEL
LIN {X 0,Y 281.719,Z 947.723,A -85,B 0,C 180,E1 -17389.69,E2 -17389.69} C_VEL
LIN {X 0,Y 283.936,Z 939.703,A -85,B 0,C 180,E1 -17391.422,E2 -17391.422} C_VEL
LIN {X 0,Y 286.727,Z 930.201,A -85,B 0,C 180,E1 -17393.098,E2 -17393.098} C_VEL
LIN {X 0,Y 289.505,Z 920.062,A -85,B 0,C 180,E1 -17394.573,E2 -17394.573} C_VEL
LIN {X 0,Y 292.306,Z 909.476,A -85,B 0,C 180,E1 -17395.843,E2 -17395.843} C_VEL
LIN {X 0,Y 295.085,Z 898.286,A -85,B 0,C 180,E1 -17396.914,E2 -17396.914} C_VEL
LIN {X 0,Y 297.769,Z 885.605,A -85,B 0,C 180,E1 -17397.888,E2 -17397.888} C_VEL
LIN {X 0,Y 300.435,Z 870.367,A -85,B 0,C 180,E1 -17398.76,E2 -17398.76} C_VEL
LIN {X 0,Y 304.079,Z 837.719,A -85,B 0,C 180,E1 -17400.16,E2 -17400.16} C_VEL
LIN {X 0,Y 304.813,Z 816.284,A -85,B 0,C 180,E1 -17401.492,E2 -17401.492} C_VEL
LIN {X 0,Y 304.766,Z 800.31,A -85,B 0,C 180,E1 -17402.738,E2 -17402.738} C_VEL
LIN {X 0,Y 304.431,Z 783.539,A -85,B 0,C 180,E1 -17404.264,E2 -17404.264} C_VEL
LIN {X 0,Y 304.064,Z 770.019,A -85,B 0,C 180,E1 -17405.675,E2 -17405.675} C_VEL
LIN {X 0,Y 302.86,Z 764.572,A -85,B 0,C 180,E1 -17406.723,E2 -17406.723} C_VEL
LIN {X 0,Y 300.686,Z 754.338,A -85,B 0,C 180,E1 -17409.138,E2 -17409.138} C_VEL
LIN {X 0,Y 299.751,Z 749.042,A -85,B 0,C 180,E1 -17410.642,E2 -17410.642} C_VEL
LIN {X 0,Y 297.868,Z 745.602,A -85,B 0,C 180,E1 -17413.32,E2 -17413.32} C_VEL
LIN {X 0,Y 297.22,Z 744.541,A -85,B 0,C 180,E1 -17415.193,E2 -17415.193} C_VEL
LIN {X 0,Y 297.209,Z 744.094,A -85,B 0,C 180,E1 -17417.151,E2 -17417.151} C_VEL
LIN {X 0,Y 298.045,Z 744.363,A -85,B 0,C 180,E1 -17419.414,E2 -17419.414} C_VEL
LIN {X 0,Y 299.994,Z 745.79,A -85,B 0,C 180,E1 -17421.792,E2 -17421.792} C_VEL
LIN {X 0,Y 301.191,Z 746.983,A -85,B 0,C 180,E1 -17422.887,E2 -17422.887} C_VEL
LIN {X 0,Y 302.934,Z 750.197,A -85,B 0,C 180,E1 -17424.392,E2 -17424.392} C_VEL
LIN {X 0,Y 303.94,Z 751.659,A -85,B 0,C 180,E1 -17425.086,E2 -17425.086} C_VEL
LIN {X 0,Y 306.725,Z 756.52,A -85,B 0,C 180,E1 -17426.828,E2 -17426.828} C_VEL
LIN {X 0,Y 310.112,Z 762.896,A -85,B 0,C 180,E1 -17428.603,E2 -17428.603} C_VEL
LIN {X 0,Y 311.489,Z 765.749,A -85,B 0,C 180,E1 -17429.249,E2 -17429.249} C_VEL
LIN {X 0,Y 307.229,Z 800.913,A -85,B 0,C 180,E1 -17430.801,E2 -17430.801} C_VEL
LIN {X 0,Y 305.524,Z 819.572,A -85,B 0,C 180,E1 -17431.802,E2 -17431.802} C_VEL
LIN {X 0,Y 304.016,Z 832.58,A -85,B 0,C 180,E1 -17432.741,E2 -17432.741} C_VEL
LIN {X 0,Y 301.95,Z 845.258,A -85,B 0,C 180,E1 -17433.939,E2 -17433.939} C_VEL
LIN {X 0,Y 300.055,Z 854.665,A -85,B 0,C 180,E1 -17435.064,E2 -17435.064} C_VEL
LIN {X 0,Y 297.882,Z 863.72,A -85,B 0,C 180,E1 -17436.354,E2 -17436.354} C_VEL
LIN {X 0,Y 295.898,Z 871.343,A -85,B 0,C 180,E1 -17437.665,E2 -17437.665} C_VEL
LIN {X 0,Y 293.951,Z 877.864,A -85,B 0,C 180,E1 -17438.984,E2 -17438.984} C_VEL
LIN {X 0,Y 291.638,Z 884.723,A -85,B 0,C 180,E1 -17440.649,E2 -17440.649} C_VEL
LIN {X 0,Y 289.526,Z 890.463,A -85,B 0,C 180,E1 -17442.336,E2 -17442.336} C_VEL
LIN {X 0,Y 287.195,Z 895.999,A -85,B 0,C 180,E1 -17444.384,E2 -17444.384} C_VEL
LIN {X 0,Y 285.03,Z 900.314,A -85,B 0,C 180,E1 -17446.453,E2 -17446.453} C_VEL
LIN {X 0,Y 284.438,Z 901.577,A -85,B 0,C 180,E1 -17447.151,E2 -17447.151} C_VEL
LIN {X 0,Y 282.09,Z 905.045,A -85,B 0,C 180,E1 -17449.956,E2 -17449.956} C_VEL
LIN {X 0,Y 281.122,Z 906.187,A -85,B 0,C 180,E1 -17451.373,E2 -17451.373} C_VEL
LIN {X 0,Y 279.685,Z 906.968,A -85,B 0,C 180,E1 -17454.231,E2 -17454.231} C_VEL
LIN {X 0,Y 279.167,Z 906.737,A -85,B 0,C 180,E1 -17455.669,E2 -17455.669} C_VEL
LIN {X 0,Y 278.55,Z 906.071,A -85,B 0,C 180,E1 -17457.108,E2 -17457.108} C_VEL
LIN {X 0,Y 278.227,Z 904.894,A -85,B 0,C 180,E1 -17458.553,E2 -17458.553} C_VEL
LIN {X 0,Y 277.682,Z 902.411,A -85,B 0,C 180,E1 -17460.725,E2 -17460.725} C_VEL
LIN {X 0,Y 277.493,Z 900.263,A -85,B 0,C 180,E1 -17462.177,E2 -17462.177} C_VEL
LIN {X 0,Y 277.29,Z 895.995,A -85,B 0,C 180,E1 -17464.361,E2 -17464.361} C_VEL
LIN {X 0,Y 277.745,Z 889.393,A -85,B 0,C 180,E1 -17466.903,E2 -17466.903} C_VEL
LIN {X 0,Y 278.037,Z 883.594,A -85,B 0,C 180,E1 -17468.723,E2 -17468.723} C_VEL
LIN {X 0,Y 278.415,Z 876.664,A -85,B 0,C 180,E1 -17470.545,E2 -17470.545} C_VEL
LIN {X 0,Y 278.869,Z 870.191,A -85,B 0,C 180,E1 -17472,E2 -17472} C_VEL
LIN {X 0,Y 279.473,Z 861.618,A -85,B 0,C 180,E1 -17473.636,E2 -17473.636} C_VEL
LIN {X 0,Y 279.992,Z 852.576,A -85,B 0,C 180,E1 -17475.095,E2 -17475.095} C_VEL
LIN {X 0,Y 280.641,Z 843.227,A -85,B 0,C 180,E1 -17476.364,E2 -17476.364} C_VEL
LIN {X 0,Y 281.216,Z 833.63,A -85,B 0,C 180,E1 -17477.452,E2 -17477.452} C_VEL
LIN {X 0,Y 281.713,Z 823.609,A -85,B 0,C 180,E1 -17478.39,E2 -17478.39} C_VEL
LIN {X 0,Y 282.149,Z 813.183,A -85,B 0,C 180,E1 -17479.177,E2 -17479.177} C_VEL
LIN {X 0,Y 282.435,Z 802.225,A -85,B 0,C 180,E1 -17479.819,E2 -17479.819} C_VEL
LIN {X 0,Y 282.725,Z 788.134,A -85,B 0,C 180,E1 -17480.414,E2 -17480.414} C_VEL
LIN {X 0,Y 284.035,Z 739.957,A -85,B 0,C 180,E1 -17482.182,E2 -17482.182} C_VEL
LIN {X 0,Y 277.326,Z 717.94,A -85,B 0,C 180,E1 -17483.363,E2 -17483.363} C_VEL
LIN {X 0,Y 277.291,Z 717.94,A -85,B 0,C 180,E1 -17487.478,E2 -17487.478} C_VEL
LIN {X 0,Y 277.262,Z 717.947,A -85,B 0,C 180,E1 -17492.162,E2 -17492.162} C_VEL
LIN {X 0,Y 277.295,Z 717.94,A -85,B 0,C 180,E1 -17495.792,E2 -17495.792} C_VEL
LIN {X 0,Y 277.239,Z 717.947,A -85,B 0,C 180,E1 -17499.328,E2 -17499.328} C_VEL
LIN {X 0,Y 277.213,Z 717.95,A -85,B 0,C 180,E1 -17503.198,E2 -17503.198} C_VEL
LIN {X 0,Y 277.213,Z 717.95,A -85,B 0,C 180,E1 -17507.326,E2 -17507.326} C_VEL
LIN {X 0,Y 277.269,Z 717.941,A -85,B 0,C 180,E1 -17511.792,E2 -17511.792} C_VEL
LIN {X 0,Y 277.296,Z 717.937,A -85,B 0,C 180,E1 -17514.334,E2 -17514.334} C_VEL
LIN {X 0,Y 277.256,Z 717.944,A -85,B 0,C 180,E1 -17517.829,E2 -17517.829} C_VEL
LIN {X 0,Y 277.26,Z 717.943,A -85,B 0,C 180,E1 -17520.993,E2 -17520.993} C_VEL
LIN {X 0,Y 278.372,Z 720.96,A -85,B 0,C 180,E1 -17521.246,E2 -17521.246} C_VEL
LIN {X 0,Y 286.462,Z 736.44,A -85,B 0,C 180,E1 -17522.601,E2 -17522.601} C_VEL
LIN {X 0,Y 292.734,Z 750.261,A -85,B 0,C 180,E1 -17523.638,E2 -17523.638} C_VEL
LIN {X 0,Y 291.893,Z 792.685,A -85,B 0,C 180,E1 -17524.699,E2 -17524.699} C_VEL
LIN {X 0,Y 291.692,Z 807.691,A -85,B 0,C 180,E1 -17525.199,E2 -17525.199} C_VEL
LIN {X 0,Y 291.14,Z 820.949,A -85,B 0,C 180,E1 -17525.953,E2 -17525.953} C_VEL
LIN {X 0,Y 290.213,Z 832.464,A -85,B 0,C 180,E1 -17526.856,E2 -17526.856} C_VEL
LIN {X 0,Y 288.974,Z 844.038,A -85,B 0,C 180,E1 -17528.046,E2 -17528.046} C_VEL
LIN {X 0,Y 287.523,Z 854.502,A -85,B 0,C 180,E1 -17529.42,E2 -17529.42} C_VEL
LIN {X 0,Y 285.992,Z 864.097,A -85,B 0,C 180,E1 -17530.989,E2 -17530.989} C_VEL
LIN {X 0,Y 284.568,Z 872.789,A -85,B 0,C 180,E1 -17532.752,E2 -17532.752} C_VEL
LIN {X 0,Y 282.829,Z 881.291,A -85,B 0,C 180,E1 -17534.867,E2 -17534.867} C_VEL
LIN {X 0,Y 281.354,Z 888.051,A -85,B 0,C 180,E1 -17536.999,E2 -17536.999} C_VEL
LIN {X 0,Y 280.418,Z 893.415,A -85,B 0,C 180,E1 -17539.157,E2 -17539.157} C_VEL
LIN {X 0,Y 279.822,Z 896.35,A -85,B 0,C 180,E1 -17540.595,E2 -17540.595} C_VEL
LIN {X 0,Y 278.747,Z 899.91,A -85,B 0,C 180,E1 -17542.749,E2 -17542.749} C_VEL
LIN {X 0,Y 278.306,Z 901.732,A -85,B 0,C 180,E1 -17544.193,E2 -17544.193} C_VEL
LIN {X 0,Y 278.004,Z 904.042,A -85,B 0,C 180,E1 -17547.092,E2 -17547.092} C_VEL
LIN {X 0,Y 277.749,Z 904.882,A -85,B 0,C 180,E1 -17549.99,E2 -17549.99} C_VEL
LIN {X 0,Y 278,Z 904.117,A -85,B 0,C 180,E1 -17552.888,E2 -17552.888} C_VEL
LIN {X 0,Y 278.287,Z 901.886,A -85,B 0,C 180,E1 -17555.788,E2 -17555.788} C_VEL
LIN {X 0,Y 279.03,Z 899.068,A -85,B 0,C 180,E1 -17557.953,E2 -17557.953} C_VEL
LIN {X 0,Y 280.041,Z 895.239,A -85,B 0,C 180,E1 -17560.107,E2 -17560.107} C_VEL
LIN {X 0,Y 281.104,Z 889.765,A -85,B 0,C 180,E1 -17562.487,E2 -17562.487} C_VEL
LIN {X 0,Y 282.535,Z 882.951,A -85,B 0,C 180,E1 -17564.761,E2 -17564.761} C_VEL
LIN {X 0,Y 284.206,Z 874.92,A -85,B 0,C 180,E1 -17566.88,E2 -17566.88} C_VEL
LIN {X 0,Y 285.675,Z 866.699,A -85,B 0,C 180,E1 -17568.641,E2 -17568.641} C_VEL
LIN {X 0,Y 287.26,Z 856.526,A -85,B 0,C 180,E1 -17570.392,E2 -17570.392} C_VEL
LIN {X 0,Y 288.813,Z 846.052,A -85,B 0,C 180,E1 -17571.82,E2 -17571.82} C_VEL
LIN {X 0,Y 290.121,Z 834.779,A -85,B 0,C 180,E1 -17573.042,E2 -17573.042} C_VEL
LIN {X 0,Y 291.18,Z 822.844,A -85,B 0,C 180,E1 -17574.023,E2 -17574.023} C_VEL
LIN {X 0,Y 291.683,Z 810.612,A -85,B 0,C 180,E1 -17574.771,E2 -17574.771} C_VEL
LIN {X 0,Y 291.939,Z 797.919,A -85,B 0,C 180,E1 -17575.271,E2 -17575.271} C_VEL
LIN {X 0,Y 292.716,Z 755.63,A -85,B 0,C 180,E1 -17576.341,E2 -17576.341} C_VEL
LIN {X 0,Y 292.694,Z 750.096,A -85,B 0,C 180,E1 -17576.493,E2 -17576.493} C_VEL
LIN {X 0,Y 284.658,Z 732.718,A -85,B 0,C 180,E1 -17577.826,E2 -17577.826} C_VEL
LIN {X 0,Y 278.4,Z 721.004,A -85,B 0,C 180,E1 -17578.877,E2 -17578.877} C_VEL
LIN {X 0,Y 277.305,Z 718.163,A -85,B 0,C 180,E1 -17579.09,E2 -17579.09} C_VEL
LIN {X 0,Y 277.287,Z 717.941,A -85,B 0,C 180,E1 -17579.266,E2 -17579.266} C_VEL
LIN {X 0,Y 277.223,Z 717.95,A -85,B 0,C 180,E1 -17583.885,E2 -17583.885} C_VEL
LIN {X 0,Y 277.251,Z 717.933,A -85,B 0,C 180,E1 -17587.457,E2 -17587.457} C_VEL
LIN {X 0,Y 277.256,Z 717.953,A -85,B 0,C 180,E1 -17591.212,E2 -17591.212} C_VEL
LIN {X 0,Y 277.245,Z 717.924,A -85,B 0,C 180,E1 -17595.2,E2 -17595.2} C_VEL
LIN {X 0,Y 277.249,Z 717.954,A -85,B 0,C 180,E1 -17599.486,E2 -17599.486} C_VEL
LIN {X 0,Y 277.253,Z 717.946,A -85,B 0,C 180,E1 -17603.919,E2 -17603.919} C_VEL
LIN {X 0,Y 277.192,Z 717.955,A -85,B 0,C 180,E1 -17607.829,E2 -17607.829} C_VEL
LIN {X 0,Y 277.182,Z 717.948,A -85,B 0,C 180,E1 -17610.192,E2 -17610.192} C_VEL
LIN {X 0,Y 276.511,Z 718.03,A -85,B 0,C 180,E1 -17611.405,E2 -17611.405} C_VEL
LIN {X 0,Y 273.654,Z 718.395,A -85,B 0,C 180,E1 -17613.381,E2 -17613.381} C_VEL
LIN {X 0,Y 271.241,Z 718.692,A -85,B 0,C 180,E1 -17614.986,E2 -17614.986} C_VEL
LIN {X 0,Y 270.219,Z 718.814,A -85,B 0,C 180,E1 -17616.231,E2 -17616.231} C_VEL
LIN {X 0,Y 270.143,Z 718.823,A -85,B 0,C 180,E1 -17616.653,E2 -17616.653} C_VEL
LIN {X 0,Y 270.241,Z 718.822,A -85,B 0,C 180,E1 -17620.24,E2 -17620.24} C_VEL
LIN {X 0,Y 270.333,Z 718.811,A -85,B 0,C 180,E1 -17624.931,E2 -17624.931} C_VEL
LIN {X 0,Y 270.377,Z 718.791,A -85,B 0,C 180,E1 -17629.516,E2 -17629.516} C_VEL
LIN {X 0,Y 270.54,Z 718.789,A -85,B 0,C 180,E1 -17632.537,E2 -17632.537} C_VEL
LIN {X 0,Y 270.726,Z 718.763,A -85,B 0,C 180,E1 -17638.512,E2 -17638.512} C_VEL
LIN {X 0,Y 270.726,Z 718.757,A -85,B 0,C 180,E1 -17641.487,E2 -17641.487} C_VEL
LIN {X 0,Y 270.539,Z 718.783,A -85,B 0,C 180,E1 -17647.463,E2 -17647.463} C_VEL
LIN {X 0,Y 270.377,Z 718.8,A -85,B 0,C 180,E1 -17650.484,E2 -17650.484} C_VEL
LIN {X 0,Y 270.333,Z 718.812,A -85,B 0,C 180,E1 -17655.069,E2 -17655.069} C_VEL
LIN {X 0,Y 270.239,Z 718.813,A -85,B 0,C 180,E1 -17659.76,E2 -17659.76} C_VEL
LIN {X 0,Y 270.215,Z 718.821,A -85,B 0,C 180,E1 -17664.591,E2 -17664.591} C_VEL
LIN {X 0,Y 270.214,Z 718.825,A -85,B 0,C 180,E1 -17667.915,E2 -17667.915} C_VEL
LIN {X 0,Y 270.131,Z 718.83,A -85,B 0,C 180,E1 -17671.355,E2 -17671.355} C_VEL
LIN {X 0,Y 270.164,Z 718.828,A -85,B 0,C 180,E1 -17674.911,E2 -17674.911} C_VEL
LIN {X 0,Y 270.175,Z 718.808,A -85,B 0,C 180,E1 -17678.725,E2 -17678.725} C_VEL
LIN {X 0,Y 270.211,Z 718.824,A -85,B 0,C 180,E1 -17682.551,E2 -17682.551} C_VEL
LIN {X 0,Y 270.221,Z 718.971,A -85,B 0,C 180,E1 -17686.963,E2 -17686.963} C_VEL
LIN {X 0,Y 273.272,Z 729.831,A -85,B 0,C 180,E1 -17690.492,E2 -17690.492} C_VEL
LIN {X 0,Y 275.949,Z 741.058,A -85,B 0,C 180,E1 -17693.859,E2 -17693.859} C_VEL
LIN {X 0,Y 278.383,Z 752.884,A -85,B 0,C 180,E1 -17697.189,E2 -17697.189} C_VEL
LIN {X 0,Y 278.671,Z 754.513,A -85,B 0,C 180,E1 -17697.632,E2 -17697.632} C_VEL
LIN {X 0,Y 277.376,Z 762.522,A -85,B 0,C 180,E1 -17699.566,E2 -17699.566} C_VEL
LIN {X 0,Y 276.924,Z 765.385,A -85,B 0,C 180,E1 -17700.257,E2 -17700.257} C_VEL
LIN {X 0,Y 280.827,Z 796.037,A -85,B 0,C 180,E1 -17701.585,E2 -17701.585} C_VEL
LIN {X 0,Y 283.941,Z 829.31,A -85,B 0,C 180,E1 -17702.833,E2 -17702.833} C_VEL
LIN {X 0,Y 284.361,Z 836.511,A -85,B 0,C 180,E1 -17703.073,E2 -17703.073} C_VEL
LIN {X 0,Y 283.05,Z 877.735,A -85,B 0,C 180,E1 -17704.132,E2 -17704.132} C_VEL
LIN {X 0,Y 282.003,Z 891.326,A -85,B 0,C 180,E1 -17704.763,E2 -17704.763} C_VEL
LIN {X 0,Y 280.613,Z 903.583,A -85,B 0,C 180,E1 -17705.603,E2 -17705.603} C_VEL
LIN {X 0,Y 278.894,Z 914.74,A -85,B 0,C 180,E1 -17706.628,E2 -17706.628} C_VEL
LIN {X 0,Y 276.861,Z 926.393,A -85,B 0,C 180,E1 -17708.023,E2 -17708.023} C_VEL
LIN {X 0,Y 274.819,Z 936.915,A -85,B 0,C 180,E1 -17709.62,E2 -17709.62} C_VEL
LIN {X 0,Y 273.172,Z 945.57,A -85,B 0,C 180,E1 -17711.252,E2 -17711.252} C_VEL
LIN {X 0,Y 271.724,Z 953.75,A -85,B 0,C 180,E1 -17713.134,E2 -17713.134} C_VEL
LIN {X 0,Y 270.423,Z 961.487,A -85,B 0,C 180,E1 -17715.333,E2 -17715.333} C_VEL
LIN {X 0,Y 269.457,Z 968.815,A -85,B 0,C 180,E1 -17717.967,E2 -17717.967} C_VEL
LIN {X 0,Y 269.111,Z 973.744,A -85,B 0,C 180,E1 -17720.237,E2 -17720.237} C_VEL
LIN {X 0,Y 269.186,Z 978.002,A -85,B 0,C 180,E1 -17722.803,E2 -17722.803} C_VEL
LIN {X 0,Y 269.501,Z 981.051,A -85,B 0,C 180,E1 -17725.523,E2 -17725.523} C_VEL
LIN {X 0,Y 269.67,Z 982.124,A -85,B 0,C 180,E1 -17727.022,E2 -17727.022} C_VEL
LIN {X 0,Y 269.829,Z 982.785,A -85,B 0,C 180,E1 -17728.517,E2 -17728.517} C_VEL
LIN {X 0,Y 269.983,Z 983.028,A -85,B 0,C 180,E1 -17730.01,E2 -17730.01} C_VEL
LIN {X 0,Y 269.828,Z 982.77,A -85,B 0,C 180,E1 -17731.502,E2 -17731.502} C_VEL
LIN {X 0,Y 269.668,Z 982.098,A -85,B 0,C 180,E1 -17732.998,E2 -17732.998} C_VEL
LIN {X 0,Y 269.491,Z 981.012,A -85,B 0,C 180,E1 -17734.497,E2 -17734.497} C_VEL
LIN {X 0,Y 269.156,Z 978.034,A -85,B 0,C 180,E1 -17737.146,E2 -17737.146} C_VEL
LIN {X 0,Y 269.417,Z 970.641,A -85,B 0,C 180,E1 -17742.055,E2 -17742.055} C_VEL
LIN {X 0,Y 270.275,Z 966.07,A -85,B 0,C 180,E1 -17744.311,E2 -17744.311} C_VEL
LIN {X 0,Y 271.751,Z 959.38,A -85,B 0,C 180,E1 -17746.885,E2 -17746.885} C_VEL
LIN {X 0,Y 273.868,Z 952.134,A -85,B 0,C 180,E1 -17749.107,E2 -17749.107} C_VEL
LIN {X 0,Y 275.948,Z 945.143,A -85,B 0,C 180,E1 -17750.898,E2 -17750.898} C_VEL
LIN {X 0,Y 278.47,Z 936.919,A -85,B 0,C 180,E1 -17752.645,E2 -17752.645} C_VEL
LIN {X 0,Y 281.179,Z 928.367,A -85,B 0,C 180,E1 -17754.169,E2 -17754.169} C_VEL
LIN {X 0,Y 284.213,Z 918.268,A -85,B 0,C 180,E1 -17755.65,E2 -17755.65} C_VEL
LIN {X 0,Y 287.252,Z 907.636,A -85,B 0,C 180,E1 -17756.921,E2 -17756.921} C_VEL
LIN {X 0,Y 290.141,Z 896.604,A -85,B 0,C 180,E1 -17757.998,E2 -17757.998} C_VEL
LIN {X 0,Y 293.252,Z 883.028,A -85,B 0,C 180,E1 -17759.041,E2 -17759.041} C_VEL
LIN {X 0,Y 296.057,Z 867.506,A -85,B 0,C 180,E1 -17759.91,E2 -17759.91} C_VEL
LIN {X 0,Y 299.535,Z 838.619,A -85,B 0,C 180,E1 -17761.191,E2 -17761.191} C_VEL
LIN {X 0,Y 300.537,Z 818.109,A -85,B 0,C 180,E1 -17762.508,E2 -17762.508} C_VEL
LIN {X 0,Y 300.733,Z 803.723,A -85,B 0,C 180,E1 -17763.654,E2 -17763.654} C_VEL
LIN {X 0,Y 300.749,Z 784.142,A -85,B 0,C 180,E1 -17765.492,E2 -17765.492} C_VEL
LIN {X 0,Y 300.604,Z 773.521,A -85,B 0,C 180,E1 -17766.681,E2 -17766.681} C_VEL
LIN {X 0,Y 298.994,Z 765.161,A -85,B 0,C 180,E1 -17768.507,E2 -17768.507} C_VEL
LIN {X 0,Y 297.749,Z 757.109,A -85,B 0,C 180,E1 -17770.598,E2 -17770.598} C_VEL
LIN {X 0,Y 297.524,Z 755.37,A -85,B 0,C 180,E1 -17771.111,E2 -17771.111} C_VEL
LIN {X 0,Y 296.035,Z 752.377,A -85,B 0,C 180,E1 -17773.518,E2 -17773.518} C_VEL
LIN {X 0,Y 295.437,Z 751.309,A -85,B 0,C 180,E1 -17775.542,E2 -17775.542} C_VEL
LIN {X 0,Y 295.804,Z 750.983,A -85,B 0,C 180,E1 -17778.298,E2 -17778.298} C_VEL
LIN {X 0,Y 297.406,Z 751.995,A -85,B 0,C 180,E1 -17780.934,E2 -17780.934} C_VEL
LIN {X 0,Y 298.955,Z 753.541,A -85,B 0,C 180,E1 -17782.534,E2 -17782.534} C_VEL
LIN {X 0,Y 300.906,Z 757.037,A -85,B 0,C 180,E1 -17784.274,E2 -17784.274} C_VEL
LIN {X 0,Y 303.819,Z 762.29,A -85,B 0,C 180,E1 -17786.277,E2 -17786.277} C_VEL
LIN {X 0,Y 306.829,Z 768.316,A -85,B 0,C 180,E1 -17788.007,E2 -17788.007} C_VEL
LIN {X 0,Y 307.306,Z 769.334,A -85,B 0,C 180,E1 -17788.264,E2 -17788.264} C_VEL
LIN {X 0,Y 302.549,Z 806.24,A -85,B 0,C 180,E1 -17789.947,E2 -17789.947} C_VEL
LIN {X 0,Y 300.74,Z 824.687,A -85,B 0,C 180,E1 -17791.041,E2 -17791.041} C_VEL
LIN {X 0,Y 299.07,Z 836.526,A -85,B 0,C 180,E1 -17791.966,E2 -17791.966} C_VEL
LIN {X 0,Y 296.956,Z 847.65,A -85,B 0,C 180,E1 -17793.088,E2 -17793.088} C_VEL
LIN {X 0,Y 294.933,Z 856.907,A -85,B 0,C 180,E1 -17794.222,E2 -17794.222} C_VEL
LIN {X 0,Y 292.617,Z 865.782,A -85,B 0,C 180,E1 -17795.524,E2 -17795.524} C_VEL
LIN {X 0,Y 290.414,Z 873.363,A -85,B 0,C 180,E1 -17796.881,E2 -17796.881} C_VEL
LIN {X 0,Y 287.859,Z 881.097,A -85,B 0,C 180,E1 -17798.517,E2 -17798.517} C_VEL
LIN {X 0,Y 285.448,Z 887.633,A -85,B 0,C 180,E1 -17800.212,E2 -17800.212} C_VEL
LIN {X 0,Y 283.185,Z 893.031,A -85,B 0,C 180,E1 -17801.927,E2 -17801.927} C_VEL
LIN {X 0,Y 281.517,Z 896.705,A -85,B 0,C 180,E1 -17803.316,E2 -17803.316} C_VEL
LIN {X 0,Y 279.936,Z 899.898,A -85,B 0,C 180,E1 -17804.716,E2 -17804.716} C_VEL
LIN {X 0,Y 277.79,Z 903.544,A -85,B 0,C 180,E1 -17806.839,E2 -17806.839} C_VEL
LIN {X 0,Y 276.506,Z 905.338,A -85,B 0,C 180,E1 -17808.268,E2 -17808.268} C_VEL
LIN {X 0,Y 274.268,Z 907.705,A -85,B 0,C 180,E1 -17811.156,E2 -17811.156} C_VEL
LIN {X 0,Y 272.742,Z 908.269,A -85,B 0,C 180,E1 -17814.084,E2 -17814.084} C_VEL
LIN {X 0,Y 272.197,Z 907.869,A -85,B 0,C 180,E1 -17815.558,E2 -17815.558} C_VEL
LIN {X 0,Y 271.548,Z 907.076,A -85,B 0,C 180,E1 -17817.033,E2 -17817.033} C_VEL
LIN {X 0,Y 271.193,Z 905.761,A -85,B 0,C 180,E1 -17818.515,E2 -17818.515} C_VEL
LIN {X 0,Y 270.644,Z 903.086,A -85,B 0,C 180,E1 -17820.744,E2 -17820.744} C_VEL
LIN {X 0,Y 270.272,Z 899.357,A -85,B 0,C 180,E1 -17822.981,E2 -17822.981} C_VEL
LIN {X 0,Y 270.33,Z 894.481,A -85,B 0,C 180,E1 -17825.221,E2 -17825.221} C_VEL
LIN {X 0,Y 270.673,Z 889.453,A -85,B 0,C 180,E1 -17827.085,E2 -17827.085} C_VEL
LIN {X 0,Y 271,Z 883.424,A -85,B 0,C 180,E1 -17828.952,E2 -17828.952} C_VEL
LIN {X 0,Y 271.388,Z 876.227,A -85,B 0,C 180,E1 -17830.822,E2 -17830.822} C_VEL
LIN {X 0,Y 271.873,Z 869.467,A -85,B 0,C 180,E1 -17832.314,E2 -17832.314} C_VEL
LIN {X 0,Y 272.53,Z 860.55,A -85,B 0,C 180,E1 -17833.991,E2 -17833.991} C_VEL
LIN {X 0,Y 273.062,Z 851.098,A -85,B 0,C 180,E1 -17835.488,E2 -17835.488} C_VEL
LIN {X 0,Y 273.903,Z 839.781,A -85,B 0,C 180,E1 -17836.97,E2 -17836.97} C_VEL
LIN {X 0,Y 274.596,Z 825.962,A -85,B 0,C 180,E1 -17838.384,E2 -17838.384} C_VEL
LIN {X 0,Y 275.097,Z 814.383,A -85,B 0,C 180,E1 -17839.3,E2 -17839.3} C_VEL
LIN {X 0,Y 275.397,Z 802.688,A -85,B 0,C 180,E1 -17840.006,E2 -17840.006} C_VEL
LIN {X 0,Y 275.77,Z 785.129,A -85,B 0,C 180,E1 -17840.757,E2 -17840.757} C_VEL
LIN {X 0,Y 277.059,Z 741.221,A -85,B 0,C 180,E1 -17842.428,E2 -17842.428} C_VEL
LIN {X 0,Y 270.28,Z 718.817,A -85,B 0,C 180,E1 -17843.651,E2 -17843.651} C_VEL
LIN {X 0,Y 270.219,Z 718.821,A -85,B 0,C 180,E1 -17847.915,E2 -17847.915} C_VEL
LIN {X 0,Y 270.194,Z 718.828,A -85,B 0,C 180,E1 -17851.347,E2 -17851.347} C_VEL
LIN {X 0,Y 270.221,Z 718.826,A -85,B 0,C 180,E1 -17854.903,E2 -17854.903} C_VEL
LIN {X 0,Y 270.223,Z 718.821,A -85,B 0,C 180,E1 -17858.706,E2 -17858.706} C_VEL
LIN {X 0,Y 270.17,Z 718.826,A -85,B 0,C 180,E1 -17863.24,E2 -17863.24} C_VEL
LIN {X 0,Y 270.172,Z 718.826,A -85,B 0,C 180,E1 -17867.432,E2 -17867.432} C_VEL
LIN {X 0,Y 270.199,Z 718.82,A -85,B 0,C 180,E1 -17871.363,E2 -17871.363} C_VEL
LIN {X 0,Y 270.217,Z 718.818,A -85,B 0,C 180,E1 -17875.088,E2 -17875.088} C_VEL
LIN {X 0,Y 270.191,Z 718.823,A -85,B 0,C 180,E1 -17879.135,E2 -17879.135} C_VEL
LIN {X 0,Y 270.25,Z 718.817,A -85,B 0,C 180,E1 -17880.165,E2 -17880.165} C_VEL
LIN {X 0,Y 271.329,Z 721.81,A -85,B 0,C 180,E1 -17880.417,E2 -17880.417} C_VEL
LIN {X 0,Y 279.548,Z 737.306,A -85,B 0,C 180,E1 -17881.856,E2 -17881.856} C_VEL
LIN {X 0,Y 286.411,Z 752.238,A -85,B 0,C 180,E1 -17883.036,E2 -17883.036} C_VEL
LIN {X 0,Y 285.506,Z 792.624,A -85,B 0,C 180,E1 -17884.061,E2 -17884.061} C_VEL
LIN {X 0,Y 285.357,Z 807.399,A -85,B 0,C 180,E1 -17884.551,E2 -17884.551} C_VEL
LIN {X 0,Y 284.892,Z 819.36,A -85,B 0,C 180,E1 -17885.196,E2 -17885.196} C_VEL
LIN {X 0,Y 283.865,Z 832.397,A -85,B 0,C 180,E1 -17886.201,E2 -17886.201} C_VEL
LIN {X 0,Y 282.635,Z 843.907,A -85,B 0,C 180,E1 -17887.386,E2 -17887.386} C_VEL
LIN {X 0,Y 281.09,Z 854.339,A -85,B 0,C 180,E1 -17888.735,E2 -17888.735} C_VEL
LIN {X 0,Y 279.716,Z 863.168,A -85,B 0,C 180,E1 -17890.164,E2 -17890.164} C_VEL
LIN {X 0,Y 278.166,Z 872.204,A -85,B 0,C 180,E1 -17891.962,E2 -17891.962} C_VEL
LIN {X 0,Y 276.311,Z 880.986,A -85,B 0,C 180,E1 -17894.123,E2 -17894.123} C_VEL
LIN {X 0,Y 274.628,Z 888.655,A -85,B 0,C 180,E1 -17896.523,E2 -17896.523} C_VEL
LIN {X 0,Y 273.519,Z 894.419,A -85,B 0,C 180,E1 -17898.88,E2 -17898.88} C_VEL
LIN {X 0,Y 272.891,Z 897.354,A -85,B 0,C 180,E1 -17900.354,E2 -17900.354} C_VEL
LIN {X 0,Y 271.777,Z 900.914,A -85,B 0,C 180,E1 -17902.562,E2 -17902.562} C_VEL
LIN {X 0,Y 271.315,Z 902.736,A -85,B 0,C 180,E1 -17904.043,E2 -17904.043} C_VEL
LIN {X 0,Y 270.985,Z 905.045,A -85,B 0,C 180,E1 -17907.017,E2 -17907.017} C_VEL
LIN {X 0,Y 270.722,Z 905.885,A -85,B 0,C 180,E1 -17909.99,E2 -17909.99} C_VEL
LIN {X 0,Y 270.982,Z 905.12,A -85,B 0,C 180,E1 -17912.963,E2 -17912.963} C_VEL
LIN {X 0,Y 271.295,Z 902.888,A -85,B 0,C 180,E1 -17915.937,E2 -17915.937} C_VEL
LIN {X 0,Y 272.072,Z 900.069,A -85,B 0,C 180,E1 -17918.157,E2 -17918.157} C_VEL
LIN {X 0,Y 273.125,Z 896.241,A -85,B 0,C 180,E1 -17920.366,E2 -17920.366} C_VEL
LIN {X 0,Y 274.246,Z 890.766,A -85,B 0,C 180,E1 -17922.804,E2 -17922.804} C_VEL
LIN {X 0,Y 275.744,Z 883.952,A -85,B 0,C 180,E1 -17925.133,E2 -17925.133} C_VEL
LIN {X 0,Y 277.489,Z 875.92,A -85,B 0,C 180,E1 -17927.302,E2 -17927.302} C_VEL
LIN {X 0,Y 279.025,Z 867.699,A -85,B 0,C 180,E1 -17929.102,E2 -17929.102} C_VEL
LIN {X 0,Y 280.683,Z 857.524,A -85,B 0,C 180,E1 -17930.892,E2 -17930.892} C_VEL
LIN {X 0,Y 282.3,Z 847.05,A -85,B 0,C 180,E1 -17932.35,E2 -17932.35} C_VEL
LIN {X 0,Y 283.732,Z 835.246,A -85,B 0,C 180,E1 -17933.65,E2 -17933.65} C_VEL
LIN {X 0,Y 284.815,Z 822.685,A -85,B 0,C 180,E1 -17934.683,E2 -17934.683} C_VEL
LIN {X 0,Y 285.365,Z 810.352,A -85,B 0,C 180,E1 -17935.425,E2 -17935.425} C_VEL
LIN {X 0,Y 285.606,Z 797.096,A -85,B 0,C 180,E1 -17935.929,E2 -17935.929} C_VEL
LIN {X 0,Y 286.334,Z 759.733,A -85,B 0,C 180,E1 -17936.888,E2 -17936.888} C_VEL
LIN {X 0,Y 286.404,Z 752.096,A -85,B 0,C 180,E1 -17937.093,E2 -17937.093} C_VEL
LIN {X 0,Y 278.578,Z 735.292,A -85,B 0,C 180,E1 -17938.441,E2 -17938.441} C_VEL
LIN {X 0,Y 271.289,Z 721.724,A -85,B 0,C 180,E1 -17939.721,E2 -17939.721} C_VEL
LIN {X 0,Y 270.221,Z 718.82,A -85,B 0,C 180,E1 -17939.95,E2 -17939.95} C_VEL
LIN {X 0,Y 270.189,Z 718.828,A -85,B 0,C 180,E1 -17943.657,E2 -17943.657} C_VEL
LIN {X 0,Y 270.207,Z 718.82,A -85,B 0,C 180,E1 -17946.727,E2 -17946.727} C_VEL
LIN {X 0,Y 270.23,Z 718.828,A -85,B 0,C 180,E1 -17951.043,E2 -17951.043} C_VEL
LIN {X 0,Y 270.188,Z 718.803,A -85,B 0,C 180,E1 -17955.387,E2 -17955.387} C_VEL
LIN {X 0,Y 270.203,Z 718.832,A -85,B 0,C 180,E1 -17959.439,E2 -17959.439} C_VEL
LIN {X 0,Y 270.206,Z 718.83,A -85,B 0,C 180,E1 -17963.714,E2 -17963.714} C_VEL
LIN {X 0,Y 270.152,Z 718.829,A -85,B 0,C 180,E1 -17966.885,E2 -17966.885} C_VEL
LIN {X 0,Y 270.142,Z 718.823,A -85,B 0,C 180,E1 -17970.376,E2 -17970.376} C_VEL
LIN {X 0,Y 270.203,Z 718.827,A -85,B 0,C 180,E1 -17973.757,E2 -17973.757} C_VEL
LIN {X 0,Y 270.143,Z 718.823,A -85,B 0,C 180,E1 -17976.653,E2 -17976.653} C_VEL
LIN {X 0,Y 269.493,Z 718.91,A -85,B 0,C 180,E1 -17977.897,E2 -17977.897} C_VEL
LIN {X 0,Y 266.654,Z 719.27,A -85,B 0,C 180,E1 -17979.926,E2 -17979.926} C_VEL
LIN {X 0,Y 264.261,Z 719.558,A -85,B 0,C 180,E1 -17981.576,E2 -17981.576} C_VEL
LIN {X 0,Y 263.271,Z 719.676,A -85,B 0,C 180,E1 -17982.855,E2 -17982.855} C_VEL
LIN {X 0,Y 263.211,Z 719.684,A -85,B 0,C 180,E1 -17983.287,E2 -17983.287} C_VEL
LIN {X 0,Y 263.24,Z 719.696,A -85,B 0,C 180,E1 -17986.097,E2 -17986.097} C_VEL
LIN {X 0,Y 263.457,Z 719.661,A -85,B 0,C 180,E1 -17990.79,E2 -17990.79} C_VEL
LIN {X 0,Y 263.448,Z 719.67,A -85,B 0,C 180,E1 -17993.874,E2 -17993.874} C_VEL
LIN {X 0,Y 263.692,Z 719.64,A -85,B 0,C 180,E1 -17998.473,E2 -17998.473} C_VEL
LIN {X 0,Y 263.692,Z 719.633,A -85,B 0,C 180,E1 -18001.527,E2 -18001.527} C_VEL
LIN {X 0,Y 263.502,Z 719.658,A -85,B 0,C 180,E1 -18007.664,E2 -18007.664} C_VEL
LIN {X 0,Y 263.309,Z 719.681,A -85,B 0,C 180,E1 -18010.768,E2 -18010.768} C_VEL
LIN {X 0,Y 263.281,Z 719.691,A -85,B 0,C 180,E1 -18015.482,E2 -18015.482} C_VEL
LIN {X 0,Y 263.202,Z 719.686,A -85,B 0,C 180,E1 -18020.312,E2 -18020.312} C_VEL
LIN {X 0,Y 263.15,Z 719.696,A -85,B 0,C 180,E1 -18025.297,E2 -18025.297} C_VEL
LIN {X 0,Y 263.111,Z 719.708,A -85,B 0,C 180,E1 -18028.738,E2 -18028.738} C_VEL
LIN {X 0,Y 263.081,Z 719.715,A -85,B 0,C 180,E1 -18032.295,E2 -18032.295} C_VEL
LIN {X 0,Y 263.139,Z 719.709,A -85,B 0,C 180,E1 -18035.986,E2 -18035.986} C_VEL
LIN {X 0,Y 263.115,Z 719.692,A -85,B 0,C 180,E1 -18039.871,E2 -18039.871} C_VEL
LIN {X 0,Y 263.148,Z 719.708,A -85,B 0,C 180,E1 -18043.874,E2 -18043.874} C_VEL
LIN {X 0,Y 263.151,Z 719.834,A -85,B 0,C 180,E1 -18046.145,E2 -18046.145} C_VEL
LIN {X 0,Y 266.312,Z 731.056,A -85,B 0,C 180,E1 -18049.935,E2 -18049.935} C_VEL
LIN {X 0,Y 269.176,Z 743.01,A -85,B 0,C 180,E1 -18053.642,E2 -18053.642} C_VEL
LIN {X 0,Y 271.414,Z 753.736,A -85,B 0,C 180,E1 -18056.76,E2 -18056.76} C_VEL
LIN {X 0,Y 271.772,Z 756.643,A -85,B 0,C 180,E1 -18057.562,E2 -18057.562} C_VEL
LIN {X 0,Y 270.372,Z 764.412,A -85,B 0,C 180,E1 -18059.484,E2 -18059.484} C_VEL
LIN {X 0,Y 274.528,Z 796.688,A -85,B 0,C 180,E1 -18060.92,E2 -18060.92} C_VEL
LIN {X 0,Y 277.627,Z 830.412,A -85,B 0,C 180,E1 -18062.222,E2 -18062.222} C_VEL
LIN {X 0,Y 277.977,Z 837.282,A -85,B 0,C 180,E1 -18062.453,E2 -18062.453} C_VEL
LIN {X 0,Y 276.663,Z 876.453,A -85,B 0,C 180,E1 -18063.477,E2 -18063.477} C_VEL
LIN {X 0,Y 275.567,Z 890.419,A -85,B 0,C 180,E1 -18064.137,E2 -18064.137} C_VEL
LIN {X 0,Y 274.185,Z 902.58,A -85,B 0,C 180,E1 -18064.993,E2 -18064.993} C_VEL
LIN {X 0,Y 272.377,Z 913.73,A -85,B 0,C 180,E1 -18066.034,E2 -18066.034} C_VEL
LIN {X 0,Y 270.278,Z 925.382,A -85,B 0,C 180,E1 -18067.459,E2 -18067.459} C_VEL
LIN {X 0,Y 268.166,Z 935.904,A -85,B 0,C 180,E1 -18069.091,E2 -18069.091} C_VEL
LIN {X 0,Y 266.398,Z 944.55,A -85,B 0,C 180,E1 -18070.757,E2 -18070.757} C_VEL
LIN {X 0,Y 264.749,Z 953.428,A -85,B 0,C 180,E1 -18072.873,E2 -18072.873} C_VEL
LIN {X 0,Y 263.293,Z 961.618,A -85,B 0,C 180,E1 -18075.322,E2 -18075.322} C_VEL
LIN {X 0,Y 262.448,Z 967.793,A -85,B 0,C 180,E1 -18077.641,E2 -18077.641} C_VEL
LIN {X 0,Y 262.05,Z 972.723,A -85,B 0,C 180,E1 -18079.972,E2 -18079.972} C_VEL
LIN {X 0,Y 262.116,Z 977.205,A -85,B 0,C 180,E1 -18082.778,E2 -18082.778} C_VEL
LIN {X 0,Y 262.427,Z 980.038,A -85,B 0,C 180,E1 -18085.402,E2 -18085.402} C_VEL
LIN {X 0,Y 262.613,Z 981.116,A -85,B 0,C 180,E1 -18086.942,E2 -18086.942} C_VEL
LIN {X 0,Y 262.784,Z 981.78,A -85,B 0,C 180,E1 -18088.478,E2 -18088.478} C_VEL
LIN {X 0,Y 262.949,Z 982.024,A -85,B 0,C 180,E1 -18090.01,E2 -18090.01} C_VEL
LIN {X 0,Y 262.783,Z 981.764,A -85,B 0,C 180,E1 -18091.543,E2 -18091.543} C_VEL
LIN {X 0,Y 262.61,Z 981.089,A -85,B 0,C 180,E1 -18093.078,E2 -18093.078} C_VEL
LIN {X 0,Y 262.415,Z 979.999,A -85,B 0,C 180,E1 -18094.618,E2 -18094.618} C_VEL
LIN {X 0,Y 262.116,Z 977.173,A -85,B 0,C 180,E1 -18097.221,E2 -18097.221} C_VEL
LIN {X 0,Y 262.408,Z 970.041,A -85,B 0,C 180,E1 -18102.382,E2 -18102.382} C_VEL
LIN {X 0,Y 263.726,Z 963.932,A -85,B 0,C 180,E1 -18105.465,E2 -18105.465} C_VEL
LIN {X 0,Y 265.346,Z 958.144,A -85,B 0,C 180,E1 -18107.742,E2 -18107.742} C_VEL
LIN {X 0,Y 267.548,Z 951.091,A -85,B 0,C 180,E1 -18109.977,E2 -18109.977} C_VEL
LIN {X 0,Y 269.881,Z 944.21,A -85,B 0,C 180,E1 -18111.792,E2 -18111.792} C_VEL
LIN {X 0,Y 272.606,Z 936.176,A -85,B 0,C 180,E1 -18113.562,E2 -18113.562} C_VEL
LIN {X 0,Y 276.163,Z 925.638,A -85,B 0,C 180,E1 -18115.441,E2 -18115.441} C_VEL
LIN {X 0,Y 279.095,Z 916.693,A -85,B 0,C 180,E1 -18116.76,E2 -18116.76} C_VEL
LIN {X 0,Y 281.912,Z 907.572,A -85,B 0,C 180,E1 -18117.876,E2 -18117.876} C_VEL
LIN {X 0,Y 285.372,Z 895.209,A -85,B 0,C 180,E1 -18119.112,E2 -18119.112} C_VEL
LIN {X 0,Y 288.413,Z 882.939,A -85,B 0,C 180,E1 -18120.079,E2 -18120.079} C_VEL
LIN {X 0,Y 291.627,Z 866.885,A -85,B 0,C 180,E1 -18121.014,E2 -18121.014} C_VEL
LIN {X 0,Y 295.22,Z 839.847,A -85,B 0,C 180,E1 -18122.253,E2 -18122.253} C_VEL
LIN {X 0,Y 296.46,Z 820.478,A -85,B 0,C 180,E1 -18123.525,E2 -18123.525} C_VEL
LIN {X 0,Y 296.91,Z 804.762,A -85,B 0,C 180,E1 -18124.824,E2 -18124.824} C_VEL
LIN {X 0,Y 297.309,Z 786.996,A -85,B 0,C 180,E1 -18126.549,E2 -18126.549} C_VEL
LIN {X 0,Y 297.432,Z 777.216,A -85,B 0,C 180,E1 -18127.696,E2 -18127.696} C_VEL
LIN {X 0,Y 295.806,Z 766.345,A -85,B 0,C 180,E1 -18130.291,E2 -18130.291} C_VEL
LIN {X 0,Y 295.274,Z 761.664,A -85,B 0,C 180,E1 -18131.675,E2 -18131.675} C_VEL
LIN {X 0,Y 294.256,Z 759.248,A -85,B 0,C 180,E1 -18133.597,E2 -18133.597} C_VEL
LIN {X 0,Y 293.665,Z 758.078,A -85,B 0,C 180,E1 -18135.895,E2 -18135.895} C_VEL
LIN {X 0,Y 294.282,Z 757.908,A -85,B 0,C 180,E1 -18138.776,E2 -18138.776} C_VEL
LIN {X 0,Y 296.024,Z 759.222,A -85,B 0,C 180,E1 -18141.351,E2 -18141.351} C_VEL
LIN {X 0,Y 296.912,Z 760.412,A -85,B 0,C 180,E1 -18142.331,E2 -18142.331} C_VEL
LIN {X 0,Y 299.039,Z 764.421,A -85,B 0,C 180,E1 -18144.313,E2 -18144.313} C_VEL
LIN {X 0,Y 301.351,Z 768.941,A -85,B 0,C 180,E1 -18145.992,E2 -18145.992} C_VEL
LIN {X 0,Y 303.356,Z 773.315,A -85,B 0,C 180,E1 -18147.274,E2 -18147.274} C_VEL
LIN {X 0,Y 299.005,Z 803.981,A -85,B 0,C 180,E1 -18148.685,E2 -18148.685} C_VEL
LIN {X 0,Y 296.851,Z 823.319,A -85,B 0,C 180,E1 -18149.795,E2 -18149.795} C_VEL
LIN {X 0,Y 295.281,Z 834.124,A -85,B 0,C 180,E1 -18150.6,E2 -18150.6} C_VEL
LIN {X 0,Y 293.066,Z 846.131,A -85,B 0,C 180,E1 -18151.73,E2 -18151.73} C_VEL
LIN {X 0,Y 290.236,Z 858.174,A -85,B 0,C 180,E1 -18153.192,E2 -18153.192} C_VEL
LIN {X 0,Y 288.068,Z 865.945,A -85,B 0,C 180,E1 -18154.339,E2 -18154.339} C_VEL
LIN {X 0,Y 285.726,Z 873.575,A -85,B 0,C 180,E1 -18155.669,E2 -18155.669} C_VEL
LIN {X 0,Y 282.929,Z 881.548,A -85,B 0,C 180,E1 -18157.355,E2 -18157.355} C_VEL
LIN {X 0,Y 280.676,Z 887.172,A -85,B 0,C 180,E1 -18158.769,E2 -18158.769} C_VEL
LIN {X 0,Y 278.291,Z 892.746,A -85,B 0,C 180,E1 -18160.451,E2 -18160.451} C_VEL
LIN {X 0,Y 276.008,Z 897.514,A -85,B 0,C 180,E1 -18162.208,E2 -18162.208} C_VEL
LIN {X 0,Y 273.423,Z 902.038,A -85,B 0,C 180,E1 -18164.342,E2 -18164.342} C_VEL
LIN {X 0,Y 271.157,Z 905.462,A -85,B 0,C 180,E1 -18166.511,E2 -18166.511} C_VEL
LIN {X 0,Y 269.83,Z 907.221,A -85,B 0,C 180,E1 -18167.973,E2 -18167.973} C_VEL
LIN {X 0,Y 267.408,Z 909.177,A -85,B 0,C 180,E1 -18170.927,E2 -18170.927} C_VEL
LIN {X 0,Y 266.571,Z 909.595,A -85,B 0,C 180,E1 -18172.425,E2 -18172.425} C_VEL
LIN {X 0,Y 265.796,Z 909.505,A -85,B 0,C 180,E1 -18173.929,E2 -18173.929} C_VEL
LIN {X 0,Y 265.222,Z 908.976,A -85,B 0,C 180,E1 -18175.44,E2 -18175.44} C_VEL
LIN {X 0,Y 264.544,Z 908.069,A -85,B 0,C 180,E1 -18176.954,E2 -18176.954} C_VEL
LIN {X 0,Y 264.159,Z 906.609,A -85,B 0,C 180,E1 -18178.476,E2 -18178.476} C_VEL
LIN {X 0,Y 263.576,Z 903.729,A -85,B 0,C 180,E1 -18180.764,E2 -18180.764} C_VEL
LIN {X 0,Y 263.326,Z 901.22,A -85,B 0,C 180,E1 -18182.294,E2 -18182.294} C_VEL
LIN {X 0,Y 263.159,Z 896.499,A -85,B 0,C 180,E1 -18184.596,E2 -18184.596} C_VEL
LIN {X 0,Y 263.568,Z 890.533,A -85,B 0,C 180,E1 -18186.892,E2 -18186.892} C_VEL
LIN {X 0,Y 263.889,Z 884.482,A -85,B 0,C 180,E1 -18188.809,E2 -18188.809} C_VEL
LIN {X 0,Y 264.22,Z 878.588,A -85,B 0,C 180,E1 -18190.403,E2 -18190.403} C_VEL
LIN {X 0,Y 264.621,Z 872.338,A -85,B 0,C 180,E1 -18191.878,E2 -18191.878} C_VEL
LIN {X 0,Y 265.193,Z 863.723,A -85,B 0,C 180,E1 -18193.604,E2 -18193.604} C_VEL
LIN {X 0,Y 265.792,Z 854.632,A -85,B 0,C 180,E1 -18195.136,E2 -18195.136} C_VEL
LIN {X 0,Y 266.427,Z 845.216,A -85,B 0,C 180,E1 -18196.474,E2 -18196.474} C_VEL
LIN {X 0,Y 267.026,Z 835.605,A -85,B 0,C 180,E1 -18197.619,E2 -18197.619} C_VEL
LIN {X 0,Y 267.578,Z 826.007,A -85,B 0,C 180,E1 -18198.57,E2 -18198.57} C_VEL
LIN {X 0,Y 268.026,Z 815.573,A -85,B 0,C 180,E1 -18199.412,E2 -18199.412} C_VEL
LIN {X 0,Y 268.351,Z 804.53,A -85,B 0,C 180,E1 -18200.105,E2 -18200.105} C_VEL
LIN {X 0,Y 268.689,Z 789.736,A -85,B 0,C 180,E1 -18200.778,E2 -18200.778} C_VEL
LIN {X 0,Y 270.031,Z 742.399,A -85,B 0,C 180,E1 -18202.662,E2 -18202.662} C_VEL
LIN {X 0,Y 263.248,Z 719.693,A -85,B 0,C 180,E1 -18203.921,E2 -18203.921} C_VEL
LIN {X 0,Y 263.148,Z 719.705,A -85,B 0,C 180,E1 -18208.733,E2 -18208.733} C_VEL
LIN {X 0,Y 263.151,Z 719.705,A -85,B 0,C 180,E1 -18212.286,E2 -18212.286} C_VEL
LIN {X 0,Y 263.179,Z 719.698,A -85,B 0,C 180,E1 -18215.98,E2 -18215.98} C_VEL
LIN {X 0,Y 263.116,Z 719.706,A -85,B 0,C 180,E1 -18219.871,E2 -18219.871} C_VEL
LIN {X 0,Y 263.1,Z 719.704,A -85,B 0,C 180,E1 -18223.989,E2 -18223.989} C_VEL
LIN {X 0,Y 263.102,Z 719.705,A -85,B 0,C 180,E1 -18228.412,E2 -18228.412} C_VEL
LIN {X 0,Y 263.142,Z 719.7,A -85,B 0,C 180,E1 -18232.09,E2 -18232.09} C_VEL
LIN {X 0,Y 263.173,Z 719.697,A -85,B 0,C 180,E1 -18235.879,E2 -18235.879} C_VEL
LIN {X 0,Y 263.151,Z 719.7,A -85,B 0,C 180,E1 -18239.275,E2 -18239.275} C_VEL
LIN {X 0,Y 264.268,Z 722.719,A -85,B 0,C 180,E1 -18239.535,E2 -18239.535} C_VEL
LIN {X 0,Y 267.069,Z 727.561,A -85,B 0,C 180,E1 -18240.051,E2 -18240.051} C_VEL
LIN {X 0,Y 276.207,Z 745.376,A -85,B 0,C 180,E1 -18241.705,E2 -18241.705} C_VEL
LIN {X 0,Y 280.14,Z 754.209,A -85,B 0,C 180,E1 -18242.408,E2 -18242.408} C_VEL
LIN {X 0,Y 279.202,Z 793.699,A -85,B 0,C 180,E1 -18243.432,E2 -18243.432} C_VEL
LIN {X 0,Y 279.004,Z 808.824,A -85,B 0,C 180,E1 -18243.946,E2 -18243.946} C_VEL
LIN {X 0,Y 278.451,Z 821.686,A -85,B 0,C 180,E1 -18244.683,E2 -18244.683} C_VEL
LIN {X 0,Y 277.342,Z 834.483,A -85,B 0,C 180,E1 -18245.714,E2 -18245.714} C_VEL
LIN {X 0,Y 275.987,Z 846.054,A -85,B 0,C 180,E1 -18246.955,E2 -18246.955} C_VEL
LIN {X 0,Y 274.409,Z 856.515,A -85,B 0,C 180,E1 -18248.389,E2 -18248.389} C_VEL
LIN {X 0,Y 272.742,Z 866.109,A -85,B 0,C 180,E1 -18250.027,E2 -18250.027} C_VEL
LIN {X 0,Y 271.176,Z 874.8,A -85,B 0,C 180,E1 -18251.871,E2 -18251.871} C_VEL
LIN {X 0,Y 269.286,Z 883.3,A -85,B 0,C 180,E1 -18254.086,E2 -18254.086} C_VEL
LIN {X 0,Y 267.677,Z 890.06,A -85,B 0,C 180,E1 -18256.322,E2 -18256.322} C_VEL
LIN {X 0,Y 266.626,Z 895.423,A -85,B 0,C 180,E1 -18258.589,E2 -18258.589} C_VEL
LIN {X 0,Y 265.965,Z 898.358,A -85,B 0,C 180,E1 -18260.1,E2 -18260.1} C_VEL
LIN {X 0,Y 264.81,Z 901.917,A -85,B 0,C 180,E1 -18262.365,E2 -18262.365} C_VEL
LIN {X 0,Y 264.325,Z 903.739,A -85,B 0,C 180,E1 -18263.885,E2 -18263.885} C_VEL
LIN {X 0,Y 263.968,Z 906.048,A -85,B 0,C 180,E1 -18266.938,E2 -18266.938} C_VEL
LIN {X 0,Y 263.694,Z 906.888,A -85,B 0,C 180,E1 -18269.99,E2 -18269.99} C_VEL
LIN {X 0,Y 263.964,Z 906.122,A -85,B 0,C 180,E1 -18273.042,E2 -18273.042} C_VEL
LIN {X 0,Y 264.305,Z 903.891,A -85,B 0,C 180,E1 -18276.095,E2 -18276.095} C_VEL
LIN {X 0,Y 265.118,Z 901.071,A -85,B 0,C 180,E1 -18278.373,E2 -18278.373} C_VEL
LIN {X 0,Y 266.215,Z 897.242,A -85,B 0,C 180,E1 -18280.638,E2 -18280.638} C_VEL
LIN {X 0,Y 267.398,Z 891.767,A -85,B 0,C 180,E1 -18283.138,E2 -18283.138} C_VEL
LIN {X 0,Y 268.967,Z 884.952,A -85,B 0,C 180,E1 -18285.524,E2 -18285.524} C_VEL
LIN {X 0,Y 270.787,Z 876.92,A -85,B 0,C 180,E1 -18287.744,E2 -18287.744} C_VEL
LIN {X 0,Y 272.393,Z 868.698,A -85,B 0,C 180,E1 -18289.586,E2 -18289.586} C_VEL
LIN {X 0,Y 274.128,Z 858.523,A -85,B 0,C 180,E1 -18291.416,E2 -18291.416} C_VEL
LIN {X 0,Y 275.809,Z 848.049,A -85,B 0,C 180,E1 -18292.906,E2 -18292.906} C_VEL
LIN {X 0,Y 277.242,Z 836.772,A -85,B 0,C 180,E1 -18294.179,E2 -18294.179} C_VEL
LIN {X 0,Y 278.425,Z 824.828,A -85,B 0,C 180,E1 -18295.199,E2 -18295.199} C_VEL
LIN {X 0,Y 278.957,Z 812.366,A -85,B 0,C 180,E1 -18295.996,E2 -18295.996} C_VEL
LIN {X 0,Y 279.261,Z 799.017,A -85,B 0,C 180,E1 -18296.535,E2 -18296.535} C_VEL
LIN {X 0,Y 280.045,Z 760.324,A -85,B 0,C 180,E1 -18297.554,E2 -18297.554} C_VEL
LIN {X 0,Y 280.107,Z 753.961,A -85,B 0,C 180,E1 -18297.729,E2 -18297.729} C_VEL
LIN {X 0,Y 272.468,Z 737.68,A -85,B 0,C 180,E1 -18299.097,E2 -18299.097} C_VEL
LIN {X 0,Y 264.54,Z 723.131,A -85,B 0,C 180,E1 -18300.549,E2 -18300.549} C_VEL
LIN {X 0,Y 263.305,Z 720.613,A -85,B 0,C 180,E1 -18300.793,E2 -18300.793} C_VEL
LIN {X 0,Y 263.145,Z 719.705,A -85,B 0,C 180,E1 -18300.87,E2 -18300.87} C_VEL
LIN {X 0,Y 263.143,Z 719.704,A -85,B 0,C 180,E1 -18304.111,E2 -18304.111} C_VEL
LIN {X 0,Y 263.154,Z 719.685,A -85,B 0,C 180,E1 -18307.882,E2 -18307.882} C_VEL
LIN {X 0,Y 263.171,Z 719.708,A -85,B 0,C 180,E1 -18311.867,E2 -18311.867} C_VEL
LIN {X 0,Y 263.149,Z 719.684,A -85,B 0,C 180,E1 -18316.126,E2 -18316.126} C_VEL
LIN {X 0,Y 263.116,Z 719.708,A -85,B 0,C 180,E1 -18320.129,E2 -18320.129} C_VEL
LIN {X 0,Y 263.138,Z 719.707,A -85,B 0,C 180,E1 -18324.014,E2 -18324.014} C_VEL
LIN {X 0,Y 263.081,Z 719.712,A -85,B 0,C 180,E1 -18327.704,E2 -18327.704} C_VEL
LIN {X 0,Y 263.141,Z 719.696,A -85,B 0,C 180,E1 -18331.779,E2 -18331.779} C_VEL
LIN {X 0,Y 263.144,Z 719.7,A -85,B 0,C 180,E1 -18335.207,E2 -18335.207} C_VEL
LIN {X 0,Y 263.203,Z 719.698,A -85,B 0,C 180,E1 -18339.688,E2 -18339.688} C_VEL
LIN {X 0,Y 263.211,Z 719.684,A -85,B 0,C 180,E1 -18343.287,E2 -18343.287} C_VEL
LIN {X 0,Y 262.584,Z 719.773,A -85,B 0,C 180,E1 -18344.565,E2 -18344.565} C_VEL
LIN {X 0,Y 259.723,Z 720.134,A -85,B 0,C 180,E1 -18346.647,E2 -18346.647} C_VEL
LIN {X 0,Y 257.32,Z 720.422,A -85,B 0,C 180,E1 -18348.342,E2 -18348.342} C_VEL
LIN {X 0,Y 256.365,Z 720.536,A -85,B 0,C 180,E1 -18349.656,E2 -18349.656} C_VEL
LIN {X 0,Y 256.33,Z 720.542,A -85,B 0,C 180,E1 -18350.1,E2 -18350.1} C_VEL
LIN {X 0,Y 256.465,Z 720.54,A -85,B 0,C 180,E1 -18352.125,E2 -18352.125} C_VEL
LIN {X 0,Y 256.656,Z 720.516,A -85,B 0,C 180,E1 -18358.431,E2 -18358.431} C_VEL
LIN {X 0,Y 256.656,Z 720.509,A -85,B 0,C 180,E1 -18361.569,E2 -18361.569} C_VEL
LIN {X 0,Y 256.42,Z 720.547,A -85,B 0,C 180,E1 -18366.294,E2 -18366.294} C_VEL
LIN {X 0,Y 256.389,Z 720.536,A -85,B 0,C 180,E1 -18369.466,E2 -18369.466} C_VEL
LIN {X 0,Y 256.187,Z 720.572,A -85,B 0,C 180,E1 -18374.294,E2 -18374.294} C_VEL
LIN {X 0,Y 256.141,Z 720.579,A -85,B 0,C 180,E1 -18377.567,E2 -18377.567} C_VEL
LIN {X 0,Y 256.095,Z 720.57,A -85,B 0,C 180,E1 -18381.122,E2 -18381.122} C_VEL
LIN {X 0,Y 256.131,Z 720.571,A -85,B 0,C 180,E1 -18385.144,E2 -18385.144} C_VEL
LIN {X 0,Y 256.05,Z 720.583,A -85,B 0,C 180,E1 -18389.608,E2 -18389.608} C_VEL
LIN {X 0,Y 256.034,Z 720.589,A -85,B 0,C 180,E1 -18393.298,E2 -18393.298} C_VEL
LIN {X 0,Y 256.091,Z 720.573,A -85,B 0,C 180,E1 -18397.286,E2 -18397.286} C_VEL
LIN {X 0,Y 256.087,Z 720.587,A -85,B 0,C 180,E1 -18401.197,E2 -18401.197} C_VEL
LIN {X 0,Y 256.067,Z 720.595,A -85,B 0,C 180,E1 -18405.236,E2 -18405.236} C_VEL
LIN {X 0,Y 259.088,Z 731.35,A -85,B 0,C 180,E1 -18409.03,E2 -18409.03} C_VEL
LIN {X 0,Y 261.207,Z 739.753,A -85,B 0,C 180,E1 -18411.785,E2 -18411.785} C_VEL
LIN {X 0,Y 263.85,Z 751.718,A -85,B 0,C 180,E1 -18415.463,E2 -18415.463} C_VEL
LIN {X 0,Y 264.83,Z 757.179,A -85,B 0,C 180,E1 -18417.057,E2 -18417.057} C_VEL
LIN {X 0,Y 264.456,Z 760.432,A -85,B 0,C 180,E1 -18417.907,E2 -18417.907} C_VEL
LIN {X 0,Y 263.873,Z 763.576,A -85,B 0,C 180,E1 -18418.659,E2 -18418.659} C_VEL
LIN {X 0,Y 267.543,Z 791.289,A -85,B 0,C 180,E1 -18419.956,E2 -18419.956} C_VEL
LIN {X 0,Y 270.513,Z 821.499,A -85,B 0,C 180,E1 -18421.197,E2 -18421.197} C_VEL
LIN {X 0,Y 271.627,Z 837.994,A -85,B 0,C 180,E1 -18421.802,E2 -18421.802} C_VEL
LIN {X 0,Y 270.362,Z 875.289,A -85,B 0,C 180,E1 -18422.801,E2 -18422.801} C_VEL
LIN {X 0,Y 269.211,Z 888.855,A -85,B 0,C 180,E1 -18423.442,E2 -18423.442} C_VEL
LIN {X 0,Y 267.737,Z 901.569,A -85,B 0,C 180,E1 -18424.347,E2 -18424.347} C_VEL
LIN {X 0,Y 265.6,Z 914.312,A -85,B 0,C 180,E1 -18425.591,E2 -18425.591} C_VEL
LIN {X 0,Y 263.458,Z 925.675,A -85,B 0,C 180,E1 -18427.05,E2 -18427.05} C_VEL
LIN {X 0,Y 261.293,Z 935.943,A -85,B 0,C 180,E1 -18428.721,E2 -18428.721} C_VEL
LIN {X 0,Y 259.305,Z 945.238,A -85,B 0,C 180,E1 -18430.621,E2 -18430.621} C_VEL
LIN {X 0,Y 257.748,Z 953.181,A -85,B 0,C 180,E1 -18432.62,E2 -18432.62} C_VEL
LIN {X 0,Y 256.382,Z 960.599,A -85,B 0,C 180,E1 -18434.917,E2 -18434.917} C_VEL
LIN {X 0,Y 255.448,Z 966.771,A -85,B 0,C 180,E1 -18437.297,E2 -18437.297} C_VEL
LIN {X 0,Y 255.015,Z 971.704,A -85,B 0,C 180,E1 -18439.692,E2 -18439.692} C_VEL
LIN {X 0,Y 254.996,Z 975.527,A -85,B 0,C 180,E1 -18442.09,E2 -18442.09} C_VEL
LIN {X 0,Y 255.109,Z 977.514,A -85,B 0,C 180,E1 -18443.684,E2 -18443.684} C_VEL
LIN {X 0,Y 255.355,Z 979.027,A -85,B 0,C 180,E1 -18445.275,E2 -18445.275} C_VEL
LIN {X 0,Y 255.555,Z 980.108,A -85,B 0,C 180,E1 -18446.858,E2 -18446.858} C_VEL
LIN {X 0,Y 255.738,Z 980.774,A -85,B 0,C 180,E1 -18448.436,E2 -18448.436} C_VEL
LIN {X 0,Y 255.915,Z 981.021,A -85,B 0,C 180,E1 -18450.01,E2 -18450.01} C_VEL
LIN {X 0,Y 255.736,Z 980.758,A -85,B 0,C 180,E1 -18451.585,E2 -18451.585} C_VEL
LIN {X 0,Y 255.552,Z 980.081,A -85,B 0,C 180,E1 -18453.163,E2 -18453.163} C_VEL
LIN {X 0,Y 255.343,Z 978.986,A -85,B 0,C 180,E1 -18454.747,E2 -18454.747} C_VEL
LIN {X 0,Y 255.051,Z 976.355,A -85,B 0,C 180,E1 -18457.256,E2 -18457.256} C_VEL
LIN {X 0,Y 254.945,Z 973.435,A -85,B 0,C 180,E1 -18459.53,E2 -18459.53} C_VEL
LIN {X 0,Y 255.215,Z 970.521,A -85,B 0,C 180,E1 -18461.929,E2 -18461.929} C_VEL
LIN {X 0,Y 256.054,Z 966.7,A -85,B 0,C 180,E1 -18464.311,E2 -18464.311} C_VEL
LIN {X 0,Y 257.15,Z 962.397,A -85,B 0,C 180,E1 -18466.461,E2 -18466.461} C_VEL
LIN {X 0,Y 259.336,Z 955.963,A -85,B 0,C 180,E1 -18468.987,E2 -18468.987} C_VEL
LIN {X 0,Y 261.359,Z 950.178,A -85,B 0,C 180,E1 -18470.882,E2 -18470.882} C_VEL
LIN {X 0,Y 264.347,Z 941.856,A -85,B 0,C 180,E1 -18473.097,E2 -18473.097} C_VEL
LIN {X 0,Y 267.495,Z 933.757,A -85,B 0,C 180,E1 -18474.867,E2 -18474.867} C_VEL
LIN {X 0,Y 270.955,Z 924.198,A -85,B 0,C 180,E1 -18476.588,E2 -18476.588} C_VEL
LIN {X 0,Y 274.52,Z 914.112,A -85,B 0,C 180,E1 -18478.07,E2 -18478.07} C_VEL
LIN {X 0,Y 277.559,Z 904.951,A -85,B 0,C 180,E1 -18479.18,E2 -18479.18} C_VEL
LIN {X 0,Y 280.779,Z 894.137,A -85,B 0,C 180,E1 -18480.256,E2 -18480.256} C_VEL
LIN {X 0,Y 283.99,Z 882.169,A -85,B 0,C 180,E1 -18481.217,E2 -18481.217} C_VEL
LIN {X 0,Y 287.134,Z 868.341,A -85,B 0,C 180,E1 -18482.07,E2 -18482.07} C_VEL
LIN {X 0,Y 290.976,Z 843.023,A -85,B 0,C 180,E1 -18483.257,E2 -18483.257} C_VEL
LIN {X 0,Y 292.601,Z 822.468,A -85,B 0,C 180,E1 -18484.617,E2 -18484.617} C_VEL
LIN {X 0,Y 293.38,Z 807.305,A -85,B 0,C 180,E1 -18485.911,E2 -18485.911} C_VEL
LIN {X 0,Y 294.195,Z 789.455,A -85,B 0,C 180,E1 -18487.692,E2 -18487.692} C_VEL
LIN {X 0,Y 294.468,Z 781.665,A -85,B 0,C 180,E1 -18488.629,E2 -18488.629} C_VEL
LIN {X 0,Y 293.392,Z 771.696,A -85,B 0,C 180,E1 -18491.073,E2 -18491.073} C_VEL
